//冲R角定位检测																							
	IF NOT ProductPar.iModeEN.bChamferCCDEN AND NOT ProductPar.iModeEN.bEmptyRunEN AND NOT ProductPar.iModeEN.bCcdTcpEN THEN																									
		CCD_IO.boChamferPhoto:=TRUE;																								
		fRecordMouldCCDInMainPos:=arrAxisCtrl[VirAxisNo.VirMain].Status.fActPos;																								
		fRecordMouldCCDInMainPosMod:=arrAxisCtrl[VirAxisNo.VirMain].Status.fModuloActPos;																								
		TabData[TabNo.MouldPhoto].fPhotoPosM:=fDriverDDRActPos;		
		TabData[TabNo.MouldPhoto].bCCDed_M:=TRUE;		
		TabData[TabNo.MouldPhoto].bTabOffsetNG_M:=FALSE;	
		MEMSET(ADR(CCD_COM.Chamfer),0,SIZEOF(CCD_COM.Chamfer));																		
		CCD_COM.Chamfer.iFinish:=0;																								
		iAutoAuxStep4:=10;																								
	END_IF																									
//裁切定位检测																								
	IF NOT ProductPar.iModeEN.bCuterCCDEN AND NOT ProductPar.iModeEN.bEmptyRunEN AND NOT ProductPar.iModeEN.bCcdTcpEN AND TabData[TabNo.CuterPhoto].bCCDed_M THEN																									
		CCD_IO.boCuterPhoto:=TRUE;																								
		fRecordCuterCCDInMainPos:=arrAxisCtrl[VirAxisNo.VirMain].Status.fActPos;																								
		fRecordCuterCCDInMainPosMod:=arrAxisCtrl[VirAxisNo.VirMain].Status.fModuloActPos;																								
		TabData[TabNo.CuterPhoto].fPhotoPosC:=fDriverDDRActPos;
		InteData[InteNo.Cuter-2].bIntervalFail_C:=FALSE;
		TabData[TabNo.CuterPhoto].bTabOffsetNG_C:=FALSE;	
		TabData[TabNo.CuterPhoto].bCCDed_C:=TRUE;																							
		CCD_COM.Cuter.iFinish:=0;																								
		iAutoAuxStep5:=10;																								
	END_IF																									
																				
	//************************************************************************NG踢废********************************************************************************************																									
	IF  (NOT ProductPar.iModeEN.bSizeCCDEN AND BeltData[BeltNo.NGBox1+2].fPoleNGSizeNo<>30  
		AND NOT ProductPar.iModeEN.bEmptyRunEN AND NOT ProductPar.iModeEN.bCcdTcpEN ) 		 
		OR			
	 	( BeltData[BeltNo.NGBox1+2].fPoleNGSacnNo <>30 AND NOT bFlgLineScanOver AND NOT ProductPar.iModeEN.bCcdTcpEN AND NOT ProductPar.iModeEN.bLineScanCCDEN AND NOT ProductPar.iModeEN.bEmptyRunEN)  
		OR  
		(BeltData[BeltNo.NGBox1+2].bYellowMark)  OR 
         (BeltData[BeltNo.NGBox1+2].bBlueMark)  THEN	
		NG_Sum:=NG_Sum+1;
		arrCyCtrl[EvNo.	NGPushInsideAir	].Cmd.bON:=TRUE;//踢NG料打开
		arrCyCtrl[EvNo.	NGPushInsideAir	].Cmd.bOFF:=FALSE;//踢NG料关闭		
		arrCyCtrl[EVNo.NGPushInsideVacuo].Cmd.bON:=FALSE;//踢NG料真空打开
		arrCyCtrl[EVNo.NGPushInsideVacuo].Cmd.bOFF:=TRUE;//踢NG料真空关闭																	
		BeltData[BeltNo.NGBox1+2].bHavePole:=FALSE;	
		BeltData[BeltNo.NGBox1+2].stPoleNo:='';																							
	ELSE	
		arrCyCtrl[EvNo.	NGPushInsideAir	].Cmd.bON:=FALSE;//踢NG料打开
		arrCyCtrl[EvNo.	NGPushInsideAir	].Cmd.bOFF:=TRUE;//踢NG料关闭		
		arrCyCtrl[EVNo.NGPushInsideVacuo].Cmd.bON:=TRUE;//踢NG料真空打开
		arrCyCtrl[EVNo.NGPushInsideVacuo].Cmd.bOFF:=FALSE;//踢NG料真空关闭																					
	END_IF		
												
	//iNGStep:=10;
	(*IF BeltData[BeltNo.NGBox1+2].bYellowMark THEN
		Production.NGFlag[33]:=TRUE;//感应器黄标计数;
	END_IF	*)	
																
																																																																	
(*************************************************************************裁切补偿，R角补偿计算********************************************************************************************)																									
IF NOT ProductPar.iModeEN.bEmptyRunEN AND NOT ProductPar.iModeEN.bCcdTcpEN THEN				
	(*
		//////////////////////驱动辊补偿量////////////V1////////////	
	 IF  NOT   bFlgTabPosOver THEN		
			 IF TabData[TabNo.CuterPhoto+2].bCCDed_C AND NOT TabData[TabNo.CuterPhoto+2].bTabOffsetNG_C THEN
							fDriverOffset7:=TabData[TabNo.CuterPhoto+2].fTab_OffsetC-(fDriverOffsetData[1]+fDriverOffsetData[2]);
			ELSE
						   IF ABS(fDriverOffsetData[1])<0.4 THEN
								fDriverOffset7:=fDriverOffsetData[1]*0.8;
							ELSIF ABS(fDriverOffsetData[2])<0.4 THEN
								fDriverOffset7:=fDriverOffsetData[2]*0.8;
							ELSE
								fDriverOffset7:=0;
							END_IF
			 END_IF 	
			
			IF ABS(fDriverOffset7)<10 THEN
							IF ABS(fDriverOffset7)<0.6 THEN
								Polepar.fPoleWithOffset:=LIMIT(-0.35, fDriverOffset7,0.35);
							ELSE
								Polepar.fPoleWithOffset:=fDriverOffset7;  
							END_IF
			ELSE
							IF fDriverOffset7>0 THEN
								Polepar.fPoleWithOffset:=10;
							ELSIF fDriverOffset7<0 THEN
								Polepar.fPoleWithOffset:=-10;
							END_IF	
			END_IF	

	  ELSE
					 fDriverOffset7:=fDriverOffset;
					 Polepar.fPoleWithOffset:=LIMIT(-23,fDriverOffset7,23);	
	  END_IF	
	  *)
	

	  TabData[TabNo.CuterPhoto].fTab_OffsetC;  //
	  fTab_OffsetC; //裁切下个工位反馈的极耳偏移量
		//////////////////////驱动辊补偿量////////////V1////////////			
		IF TabData[TabNo.CuterPhoto+2].bCCDed_C AND NOT TabData[TabNo.CuterPhoto+2].bTabOffsetNG_C THEN
			fDriverOffset7:=TabData[TabNo.CuterPhoto+2].fTab_OffsetC-(fDriverOffsetData[1]+fDriverOffsetData[2]);
		ELSE
			IF ABS(fDriverOffsetData[1])<0.4 THEN
				fDriverOffset7:=fDriverOffsetData[1]*0.8;
			ELSIF ABS(fDriverOffsetData[2])<0.4 THEN
				fDriverOffset7:=fDriverOffsetData[2]*0.8;
			ELSE
				fDriverOffset7:=0;
			END_IF
		END_IF 		
			
			
IF NOT 	bMA1	 THEN	
	IF  NOT   bFlgTabPosOver THEN		//计算当前片下个周期补偿量   	 
				IF ABS(fDriverOffset7)<15 THEN
								IF ABS(fDriverOffset7)<1 THEN
									//bMA1:=FALSE;
									Polepar.fPoleWithOffset:=LIMIT(-0.35, fDriverOffset7,0.35);
								ELSE
									 bMA1:=TRUE;
									 iFlgCompCount:=3;
									 iCompCount:=3;
									 arrOffset[3]:=fDriverOffset7;//+fArvDriverOffsetData ;
									 arrOffset[2]:=arrOffset[1]:=fArvDriverOffsetData;	  
									//Polepar.fPoleWithOffset:=fDriverOffset7    ;  
								END_IF		
				ELSE
								iCount20:=iCount20+1;
								 IF  ABS(fDriverOffset7)>15   AND  ABS(fDriverOffset7)<30 THEN
									  iFlgCompCount:=4;
									  iCompCount:=4;
									   bMA1:=TRUE;
									  arrOffset[4]:= SEL( fDriverOffset7>0,-15,15 )  ;
		                                                         arrOffset[3]:=SEL(fDriverOffset7>0,   fDriverOffset7+15  , fDriverOffset7-15 )  ;                         
	                                                                arrOffset[2]:=arrOffset[1]:=fArvDriverOffsetData;	  
								 ELSIF ABS(fDriverOffset7)>30   AND  ABS(fDriverOffset7)<45 THEN
									   iFlgCompCount:=5;
									   iCompCount:=5;
									    bMA1:=TRUE;
									   arrOffset[5]:=SEL( fDriverOffset7>0,-15,15 ) ;
									   arrOffset[4]:=SEL( fDriverOffset7>0,-15,15 ) ;
		                                                           arrOffset[3]:=SEL(fDriverOffset7>0,   fDriverOffset7+30  , fDriverOffset7-30 )  ;       
	                                                                    arrOffset[2]:=arrOffset[1]:=fArvDriverOffsetData;	  	
		 										 
								 ELSIF ABS(fDriverOffset7)>45   AND ABS(fDriverOffset7)<60 THEN
									   iFlgCompCount:=6;		
									    iCompCount:=6;	
									     bMA1:=TRUE;
									   arrOffset[6]:=SEL( fDriverOffset7>0,-15,15 ) ;
									   arrOffset[5]:=SEL( fDriverOffset7>0,-15,15 ) ;
									   arrOffset[4]:=SEL( fDriverOffset7>0,-15,15 ) ;									   
		                                                           arrOffset[3]:=SEL(fDriverOffset7>0,   fDriverOffset7+45  , fDriverOffset7-45 )  ;    
	                                                                  arrOffset[2]:=arrOffset[1]:=fArvDriverOffsetData;	  		 
								 ELSIF ABS(fDriverOffset7)>60   AND  ABS(fDriverOffset7)<75 THEN
									   iFlgCompCount:=7;		
									   iCompCount:=7;	
                                                                          bMA1:=TRUE;	 
									   arrOffset[7]:=SEL( fDriverOffset7>0,-15,15 ) ;
									   arrOffset[6]:=SEL( fDriverOffset7>0,-15,15 ) ;
									   arrOffset[5]:=SEL( fDriverOffset7>0,-15,15 ) ;		
									   arrOffset[4]:=SEL( fDriverOffset7>0,-15,15 ) ;						   
		                                                            arrOffset[3]:=SEL(fDriverOffset7>0,   fDriverOffset7+60  , fDriverOffset7-60 )  ;    
	                                                                   arrOffset[2]:=arrOffset[1]:=fArvDriverOffsetData;										   
								ELSIF  ABS(fDriverOffset7)>75  THEN
									   iFlgCompCount:=7;		
									   iCompCount:=7;	
                                                                           bMA1:=TRUE;	 
									   arrOffset[7]:=SEL( fDriverOffset7>0,-15,15 ) ;
									   arrOffset[6]:=SEL( fDriverOffset7>0,-15,15 ) ;
									   arrOffset[5]:=SEL( fDriverOffset7>0,-15,15 ) ;		
									   arrOffset[4]:=SEL( fDriverOffset7>0,-15,15 ) ;						   
		                                                           arrOffset[3]:=SEL(fDriverOffset7>0,   fDriverOffset7+60  , fDriverOffset7-60 )  ;    
	                                                                  arrOffset[2]:=arrOffset[1]:=fArvDriverOffsetData;		      
								 END_IF
								
				END_IF	
	ELSE	
					                       fDriverOffset7:=fDriverOffset;
								 IF  ABS(fDriverOffset7)>30   AND  ABS(fDriverOffset7)<60 THEN
									  iFlgCompCount:=4;
									  iCompCount:=4;
									   bMA1:=TRUE;
									  arrOffset[4]:= SEL( fDriverOffset7>0,-30,30 )  ;
		                                                         arrOffset[3]:=SEL(fDriverOffset7>0,   fDriverOffset7+30  , fDriverOffset7-30 )  ;                         
	                                                                arrOffset[2]:=arrOffset[1]:=fArvDriverOffsetData;	  
								 ELSIF ABS(fDriverOffset7)>60   AND  ABS(fDriverOffset7)<90 THEN
									   iFlgCompCount:=5;
									   iCompCount:=5;
									    bMA1:=TRUE;
									   arrOffset[5]:=SEL( fDriverOffset7>0,-30,30 ) ;
									   arrOffset[4]:=SEL( fDriverOffset7>0,-30,30 ) ;
		                                                           arrOffset[3]:=SEL(fDriverOffset7>0,   fDriverOffset7+60  , fDriverOffset7-60 )  ;       
	                                                                    arrOffset[2]:=arrOffset[1]:=fArvDriverOffsetData;	  	
		 										 
								 ELSIF ABS(fDriverOffset7)>90   AND ABS(fDriverOffset7)<120 THEN
									   iFlgCompCount:=6;		
									    iCompCount:=6;	
									     bMA1:=TRUE;
									   arrOffset[6]:=SEL( fDriverOffset7>0,-30,30 ) ;
									   arrOffset[5]:=SEL( fDriverOffset7>0,-30,30 ) ;
									   arrOffset[4]:=SEL( fDriverOffset7>0,-30,30 ) ;									   
		                                                           arrOffset[3]:=SEL(fDriverOffset7>0,   fDriverOffset7+90  , fDriverOffset7-90 )  ;    
	                                                                  arrOffset[2]:=arrOffset[1]:=fArvDriverOffsetData;	  		 
								 ELSIF ABS(fDriverOffset7)>120   AND  ABS(fDriverOffset7)<150 THEN
									   iFlgCompCount:=7;		
									   iCompCount:=7;	
                                                                          bMA1:=TRUE;	 
									   arrOffset[7]:=SEL( fDriverOffset7>0,-30,30 ) ;
									   arrOffset[6]:=SEL( fDriverOffset7>0,-30,30 ) ;
									   arrOffset[5]:=SEL( fDriverOffset7>0,-30,30 ) ;		
									   arrOffset[4]:=SEL( fDriverOffset7>0,-30,30 ) ;						   
		                                                            arrOffset[3]:=SEL(fDriverOffset7>0,   fDriverOffset7+120  , fDriverOffset7-120 )  ;    
	                                                                   arrOffset[2]:=arrOffset[1]:=fArvDriverOffsetData;										   
								ELSIF  ABS(fDriverOffset7)>150  THEN
						                           iFlgCompCount:=7;		
									   iCompCount:=7;	
                                                                           bMA1:=TRUE;	 
									   arrOffset[7]:=SEL( fDriverOffset7>0,-30,30 ) ;
									   arrOffset[6]:=SEL( fDriverOffset7>0,-30,30 ) ;
									   arrOffset[5]:=SEL( fDriverOffset7>0,-30,30 ) ;		
									   arrOffset[4]:=SEL( fDriverOffset7>0,-30,30 ) ;						   
		                                                            arrOffset[3]:=SEL(fDriverOffset7>0,   fDriverOffset7+120  , fDriverOffset7-120 )  ;    
	                                                                   arrOffset[2]:=arrOffset[1]:=fArvDriverOffsetData;			      
								 END_IF								 
					                //Polepar.fPoleWithOffset:=LIMIT(-23,fDriverOffset7,23);	
	 END_IF		
	 
END_IF

	(************补偿大偏移量后面的极片模糊补偿 *****************)
	IF  bMA1 THEN
		 Polepar.fPoleWithOffset:=arrOffset[iCompCount]; 
		IF 	iCompCount<=1 THEN
			bMA1:=FALSE;
			iFlgCompCount:=0;
			MEMSET(ADR(arrOffset),0,SIZEOF(arrOffset));
		END_IF
	END_IF			
		
(************计算近10次补偿有效值的平均值******************)
   K2:=0;
   fSumDriverOffsetData:=0;
	FOR i30:=1 TO 10 BY 1 DO
		IF  ABS( fDriverOffsetData[i30])  <0.3   AND  ABS( fDriverOffsetData[i30])  >0  THEN 		//
			K2:=K2+1;
		    fSumDriverOffsetData:=fSumDriverOffsetData+fDriverOffsetData[i30];
		END_IF
		
		IF  i30=10   THEN
			IF K2>=1 THEN 
			   fArvDriverOffsetData:=fSumDriverOffsetData/K2;
			ELSE
			   fArvDriverOffsetData:=0;
			END_IF
		END_IF		
	END_FOR	
	

				
(*-----------20240404
//裁切补偿计算																								
IF NOT ProductPar.iModeEN.bEmptyRunEN AND NOT ProductPar.iModeEN.bCcdTcpEN AND NOT ProductPar.iModeEN.bCuterCCDEN   THEN			
	IF   ProductPar.bCompSel OR TRUE THEN	  //极耳定位补偿方式																				
	(*	IF TabData[TabNo.CuterPhoto+2].bCCDed_C AND NOT TabData[TabNo.CuterPhoto+2].bTabOffsetNG_C THEN
			fDriverOffset7:=TabData[TabNo.CuterPhoto+2].fTab_OffsetC-(fDriverOffsetData[1]+fDriverOffsetData[2]);
		ELSE
			fDriverOffset7:=0;
		END_IF*)
		
	   
	    	 IF  NOT   bFlgTabPosOver THEN
					 
						(*IF TabData[TabNo.CuterPhoto+2].bCCDed_C AND NOT TabData[TabNo.CuterPhoto+2].bTabOffsetNG_C THEN
							fDriverOffset7:=TabData[TabNo.CuterPhoto+2].fTab_OffsetC-(fDriverOffsetData[1]+fDriverOffsetData[2]);
						ELSE
						fDriverOffset7:=0;
					  END_IF*)
			 
					 IF TabData[TabNo.CuterPhoto+2].bCCDed_C AND NOT TabData[TabNo.CuterPhoto+2].bTabOffsetNG_C THEN
							fDriverOffset7:=TabData[TabNo.CuterPhoto+2].fTab_OffsetC-(fDriverOffsetData[1]+fDriverOffsetData[2]);
					  ELSE
						   IF ABS(fDriverOffsetData[1])<0.4 THEN
								fDriverOffset7:=fDriverOffsetData[1]*0.8;
							ELSIF ABS(fDriverOffsetData[2])<0.4 THEN
								fDriverOffset7:=fDriverOffsetData[2]*0.8;
							ELSE
								fDriverOffset7:=0;
							END_IF
					  END_IF 
				  
				  
				  
                   (*   IF TabData[TabNo.CuterPhoto+2].bCCDed_C AND NOT TabData[TabNo.CuterPhoto+2].bTabOffsetNG_C THEN
							
								IF TabData[TabNo.CuterPhoto+3].bCCDed_C AND NOT TabData[TabNo.CuterPhoto+3].bTabOffsetNG_C  THEN
									fDriverOffset7:=(TabData[TabNo.CuterPhoto+2].fTab_OffsetC+TabData[TabNo.CuterPhoto+3].fTab_OffsetC)/2 - (fDriverOffsetData[1]+fDriverOffsetData[2]);
							ELSE
									fDriverOffset7:=TabData[TabNo.CuterPhoto+2].fTab_OffsetC-(fDriverOffsetData[1]+fDriverOffsetData[2]);
							END_IF
						ELSE
							IF ABS(fDriverOffsetData[1])<0.4 THEN
									fDriverOffset7:=fDriverOffsetData[1]*0.8;
								ELSIF ABS(fDriverOffsetData[2])<0.4 THEN
								fDriverOffset7:=fDriverOffsetData[2]*0.8;
							ELSE
								fDriverOffset7:=0;
								END_IF
							
						END_IF 	*)
				
					
						(*	
						IF ABS(fDriverOffset7)<10 THEN
							Polepar.fPoleWithOffset:=fDriverOffset7;
						ELSE
							IF fDriverOffset7>0 THEN
								Polepar.fPoleWithOffset:=10;
							ELSIF fDriverOffset7<0 THEN
								Polepar.fPoleWithOffset:=-10;
							END_IF	
						END_IF*)
						
								
						IF ABS(fDriverOffset7)<10 THEN
							IF ABS(fDriverOffset7)<0.6 THEN
								Polepar.fPoleWithOffset:=LIMIT(-0.35, fDriverOffset7,0.35);
							ELSE
								Polepar.fPoleWithOffset:=fDriverOffset7;  
							END_IF
						ELSE
							IF fDriverOffset7>0 THEN
								Polepar.fPoleWithOffset:=10;
							ELSIF fDriverOffset7<0 THEN
								Polepar.fPoleWithOffset:=-10;
							END_IF	
						END_IF	
				 ELSE
						  fDriverOffset7:=fDriverOffset;
						  Polepar.fPoleWithOffset:=LIMIT(-23,fDriverOffset7,23);	
				END_IF				
	ELSE//尺寸检测闭环纠偏
				 IF  NOT   bFlgTabPosOver THEN
						IF  ( BeltData[BeltNo.OverHang+1].iTabNGSizeNo=1  OR  BeltData[BeltNo.OverHang+1].iTabNGSizeNo=6 )  
							AND 0<=BeltData[BeltNo.OverHang+1].fTabSite AND BeltData[BeltNo.OverHang+1].fTabSite<90 THEN
						
							fDriverOffset7:=(PolePar.TabSitebace-BeltData[BeltNo.OverHang+1].fTabSite-fDriverOffsetData[1]-fDriverOffsetData[2]);
							
							//fDriverOffset7:=(PolePar.TabSitebace-BeltData[BeltNo.OverHang+1].fTabSite-
                                                                       //         LIMIT(-2, fDriverOffsetData[1] ,2) - LIMIT(-2, fDriverOffsetData[2] ,2)  ) ;
						ELSE
							fDriverOffset7:=0;
						END_IF		
				
						IF ABS(fDriverOffset7)<0.5 THEN
							Polepar.fPoleWithOffset:=LIMIT(-0.18,fDriverOffset7,0.18);
						ELSE
							Polepar.fPoleWithOffset:=LIMIT(-25,fDriverOffset7,25);
						END_IF
				 ELSE
						  fDriverOffset7:=fDriverOffset;
						  Polepar.fPoleWithOffset:=LIMIT(-25,fDriverOffset7,25);	
				END_IF
	END_IF
----------------20240404*)			
(*																						
	//模具前计算模具X纠偏补偿量
	IF TabData[TabNo.MouldPhoto+2].bCCDed_M AND NOT TabData[TabNo.MouldPhoto+2].bTabOffsetNG_M AND NOT ProductPar.iModeEN.bMouldXOffsetEN THEN
		fMouldXOffset7:=TabData[TabNo.MouldPhoto+2].fTab_OffsetM-(fDriverOffsetData[1]+fDriverOffsetData[2]+fDriverOffsetData[3]);
	ELSE
		fMouldXOffset7:=0;
	END_IF
*)	
	//模具前计算模具X纠偏补偿量	
	
	(*
	IF TabData[TabNo.MouldPhoto+2].bCCDed_M AND NOT TabData[TabNo.MouldPhoto+2].bTabOffsetNG_M AND NOT ProductPar.iModeEN.bMouldXOffsetEN THEN
		fMouldXOffset7:=TabData[TabNo.MouldPhoto+2].fTab_OffsetM-(fDriverOffsetData[1]+fDriverOffsetData[2]+fDriverOffsetData[3]);
	ELSE
		fMouldXOffset7:=0;
	END_IF	*)
										(*****************************R角补偿****************************************)	
     IF TabData[TabNo.MouldPhoto+2].bCCDed_M AND NOT TabData[TabNo.MouldPhoto+2].bTabOffsetNG_M AND NOT ProductPar.iModeEN.bMouldXOffsetEN THEN
		fMouldXOffset7:=TabData[TabNo.MouldPhoto+2].fTab_OffsetM-
                                             ( LIMIT( -1,  fDriverOffsetData[1] ,1 ) + LIMIT( -1,  fDriverOffsetData[2] ,1)+ LIMIT( -1,  fDriverOffsetData[3] ,1)  );
	ELSE
		fMouldXOffset7:=0;
	END_IF	
	
    IF TabData[TabNo.MouldPhoto+2].bCCDed_M AND NOT TabData[TabNo.MouldPhoto+2].bTabOffsetNG_M AND NOT ProductPar.iModeEN.bMouldXOffsetEN THEN
		fMouldXOffset8:= TabData[TabNo.MouldPhoto+2].fTab_OffsetY ;
                                         
	ELSE
		
		IF  NOT TabData[TabNo.MouldPhoto+3].bTabOffsetNG_M THEN
		    fMouldXOffset8:= TabData[TabNo.MouldPhoto+3].fTab_OffsetY ;
		ELSIF NOT TabData[TabNo.MouldPhoto+4].bTabOffsetNG_M THEN
			fMouldXOffset8:= TabData[TabNo.MouldPhoto+4].fTab_OffsetY ;
		ELSE
			fMouldXOffset8:=0;
		END_IF
			
	END_IF	 
	
	
	
	
	
	IF NOT ProductPar.iModeEN.bMouldXclosureEN AND NOT bCyDDRMark THEN
		IF iRTransCompCount=1  THEN
			iRTransCompCount:=28;
			(************计算近10次R角横深有效值的平均值******************)
		   K4:=0;
		   fSumTransverData:=0;
			FOR i30:=3 TO 22 BY 1 DO
				IF iPartSelect=1 THEN//正极      2---4
					IF BeltData[i30].fPoleNGSizeNo=30 THEN
						K4:=K4+1;
						(*正极RoundedSize7为叠片侧、RoundedSize8为切刀侧，故RoundedSize7-RoundedSize8*)	
						fSumTransverData:=fSumTransverData+(BeltData[i30].RoundedSize7-BeltData[i30].RoundedSize8)/2;			
					END_IF
				ELSE//负极     1.8----3.8
					IF BeltData[i30].fPoleNGSizeNo=30 THEN
						K4:=K4+1;
						(*负极RoundedSize8为叠片侧、RoundedSize7为切刀侧，故RoundedSize8-RoundedSize7*)	
						fSumTransverData:=fSumTransverData+(BeltData[i30].RoundedSize8-BeltData[i30].RoundedSize7)/2;				
					END_IF			
				END_IF		
		
				IF  i30=22   THEN
					IF K4>=15 THEN 
					  // fArvTransverData:=fArvTransverData+LIMIT(-0.1,fSumTransverData/K4*0.3,0.1);  //(-0.25,fSumTransverData/K4*0.3,0.25)
					   fArvTransverData:=fArvTransverData+SEL( ABS(fSumTransverData/K4)>=0.1,0,LIMIT(-0.25,fSumTransverData/K4*0.3,0.25));
					ELSE
					   fArvTransverData:=0;//???
					END_IF
				END_IF		
			END_FOR		
		END_IF
		IF iRTransCompCount>=1 THEN	
			iRTransCompCount:=iRTransCompCount-1;
		END_IF
	ELSE
		iRTransCompCount:=28;
		fArvTransverData:=0;	
	END_IF

	
	
	(***************************R角纵深闭环**********************************)
	bComMode:=TRUE;
IF NOT ProductPar.iModeEN.bMouldYclosureEN AND NOT bCyDDRMark THEN
	
 IF iRTransCompCount2=1  THEN
			iRTransCompCount2:=28;
			
			(************计算近10次R角纵深有效值的平均中值******************)
		   K3:=0;
		   fSumTransverData2:=0;
	FOR i30:=3 TO 22 BY 1 DO
									
			IF NOT bComMode THEN  //纵深
				(*
				IF iPartSelect=1 THEN//正极             4.7----6.3  
					(*   V1 角纵深       正极RoundedSize3为叠片侧R角纵深    、RoundedSize4为切刀侧R角纵深 ，RoundedSize3+RoundedSize4    *)
	                 IF 4.7<=BeltData[i30].RoundedSize3   AND  BeltData[i30].RoundedSize4<=6.3 THEN 
				         fSumTransverData:=fSumTransverData+(BeltData[i30].RoundedSize3+BeltData[i30].RoundedSize4)/2;		
						 K3:=K3+1;
					END_IF				
				ELSIF  iPartSelect=2 THEN//负极        1.8----3.4
					(*   V1 角纵深       正极RoundedSize3为叠片侧R角纵深    、RoundedSize4为切刀侧R角纵深 ，RoundedSize3+RoundedSize4    *)
	                 IF 1.8<=BeltData[i30].RoundedSize3   AND  BeltData[i30].RoundedSize4<=3.4 THEN 
				         fSumTransverData:=fSumTransverData+(BeltData[i30].RoundedSize3+BeltData[i30].RoundedSize4)/2;		
						 K3:=K3+1;
					END_IF			
			   END_IF
				*)
               ;	
		   ELSE//面积
				IF iPartSelect=1 THEN//正极             C+D=32.972   
				   (*   V2角面积     正极RoundedSize1为叠片侧R角面积  、RoundedSize2为切刀侧R角面积 ，RoundedSize3+RoundedSize4    *)	
				   (* IF BeltData[i30].fPoleNGSizeNo=30   THEN 	
					    fSumTransverData2:=fSumTransverData2+( (BeltData[i30].RoundedSize1+BeltData[i30].RoundedSize2)-32.972 );	
					    K3:=K3+1;
					END_IF*)	
				    IF BeltData[i30].fPoleNGSizeNo=30   THEN 	
					    fSumTransverData2:=fSumTransverData2+(BeltData[i30].RoundedSize1+BeltData[i30].RoundedSize2);	
					    K3:=K3+1;
					END_IF					
					
				ELSIF  iPartSelect=2 THEN//负极     //C+D=11.608   //C+D=11.877
				   (*   V2角面积     正极RoundedSize1为叠片侧R角面积  、RoundedSize2为切刀侧R角面积 ，RoundedSize3+RoundedSize4    *)	
				   (* IF BeltData[i30].fPoleNGSizeNo=30THEN 	
					    fSumTransverData2:=fSumTransverData2+( (BeltData[i30].RoundedSize1+BeltData[i30].RoundedSize2)-11.877 );	
					    K3:=K3+1;
					END_IF*)		
				    IF BeltData[i30].fPoleNGSizeNo=30THEN 	
					    fSumTransverData2:=fSumTransverData2+(BeltData[i30].RoundedSize1+BeltData[i30].RoundedSize2);	
					    K3:=K3+1;
					END_IF						
				END_IF	
			END_IF
							
				IF  i30=22  THEN
					IF  iPartSelect=1 THEN//正极  
							IF K3>=15 THEN 
								IF NOT bComMode THEN  //V1 角纵深    补偿方式
									(*fArvTransverData2:=fArvTransverData2+LIMIT( -0.1,   fSumTransverData2/K3-fRSizeBase   , 0.1 )  ;*)
									;
								ELSE    //V2 角面积  补偿方式
									//fArvTransverData2:=fSumTransverData2/K3;
									//   fArvTransverData2:=fArvTransverData2+LIMIT(-0.25,fSumTransverData2/K3*0.3,0.25);
								    //fArvTransverData2:=SEL( ABS(fSumTransverData2/K3-32.972)>=1.2 ,0 ,fArvTransverData2+LIMIT(-0.1,(fSumTransverData2/K3-32.972)*0.3,0.1));
									 IF ABS(fSumTransverData2/K3-32.972)>=1.2 THEN
										fArvTransverData2:=fArvTransverData2+LIMIT(-0.1,(fSumTransverData2/K3-32.972)*0.3,0.1); 
									 END_IF
									
									
								END_IF		   
							ELSE
							   fArvTransverData2:=0;
							END_IF
					ELSIF  iPartSelect=2 THEN//负极  
								IF K3>=15 THEN 
									IF NOT bComMode THEN  //V1 角纵深    补偿方式
										(*fArvTransverData2:=fArvTransverData2+LIMIT( -0.1,   fSumTransverData2/K3-fRSizeBase   , 0.1 )  ;*)
										;
									ELSE    //V2 角面积  补偿方式
										//fArvTransverData2:=fSumTransverData2/K3;
										//   fArvTransverData2:=fArvTransverData2+LIMIT(-0.25,fSumTransverData2/K3*0.3,0.25);
										//fArvTransverData2:=SEL( ABS(fSumTransverData2/K3-11.877)>=0.55 ,0 ,fArvTransverData2+LIMIT(-0.1,(fSumTransverData2/K3-11.877)*0.3,0.1));
										IF ABS(fSumTransverData2/K3-11.877)>=0.55 THEN
											fArvTransverData2:=fArvTransverData2+LIMIT(-0.1,(fSumTransverData2/K3-11.877)*0.3,0.1);
										END_IF
									END_IF		   
							ELSE
							   fArvTransverData2:=0;
							END_IF						
					END_IF		
				END_IF	
				
		END_FOR		
			
	END_IF	
		
		IF iRTransCompCount2>=1 THEN	
			iRTransCompCount2:=iRTransCompCount2-1;
		END_IF
		
ELSE
		iRTransCompCount2:=28;
		fArvTransverData2:=0;	
END_IF
	
	
	
	
	
	
	
	IF arrAxisPar[AxisNo.MouldRectify_X].arrTargetPoint[1]-fMouldXOffset7>arrAxisPar[AxisNo.MouldRectify_X].arrTargetPoint[3] OR
		arrAxisPar[AxisNo.MouldRectify_X].arrTargetPoint[1]-fMouldXOffset7<arrAxisPar[AxisNo.MouldRectify_X].arrTargetPoint[4] AND NOT ProductPar.iModeEN.bMouldXOffsetEN 
	THEN
		Polepar.fMouldX_Offset:=arrAxisPar[AxisNo.MouldRectify_X].arrTargetPoint[1]-arrAxisCtrl[AxisNo.MouldRectify_X].Status.fSetPos;
		stAlarm.arrLightWarn[8]:=TRUE;//模具X补偿量超过纠偏电机行程
	ELSE
		Polepar.fMouldX_Offset:=fMouldXOffset7;
	END_IF
	
	//arrAxisPar[AxisNo.MouldRectify_X].arrTargetPoint[2]:=arrAxisPar[AxisNo.MouldRectify_X].arrTargetPoint[1]+fArvTransverData-Polepar.fMouldX_Offset;   //V1
	
	                            //TabData[TabNo.MouldPhoto+2].fTab_OffsetM
	//arrAxisPar[AxisNo.MouldRectify_Y].arrTargetPoint[2]:=arrAxisPar[AxisNo.MouldRectify_Y].arrTargetPoint[1]-  (TabData[TabNo.MouldPhoto+2].fTab_OffsetM + TabData[TabNo.MouldPhoto+2].fTab_OffsetM )/2     ;   //V1
								
	
(*	
  IF   NOT CutMark_R[0] THEN
	arrAxisPar[AxisNo.MouldRectify_X].arrTargetPoint[2]:=arrAxisPar[AxisNo.MouldRectify_X].arrTargetPoint[1]-Polepar.fMouldX_Offset;
  ELSE
      arrAxisPar[AxisNo.MouldRectify_X].arrTargetPoint[2]:=arrAxisPar[AxisNo.MouldRectify_X].arrTargetPoint[1];
 END_IF		
*)   //V2		


(*
  IF  ABS(   PolePar.TabSitebace-BeltData[BeltNo.OverHang+1].fTabSite )<=4    AND     BeltData[BeltNo.OverHang+1].iTabNGSizeNo=1    THEN
	arrAxisPar[AxisNo.MouldRectify_X].arrTargetPoint[2]:=arrAxisPar[AxisNo.MouldRectify_X].arrTargetPoint[1]-Polepar.fMouldX_Offset;
  ELSE
      arrAxisPar[AxisNo.MouldRectify_X].arrTargetPoint[2]:=arrAxisPar[AxisNo.MouldRectify_X].arrTargetPoint[1];
 END_IF	
*)//V3



	
ELSE
	Polepar.fPoleWithOffset:=0;
	Polepar.fMouldX_Offset:=0;
END_IF	
																						
//记录模具，切刀当前的凸轮																								
	iMouldRunTableSel:=fbMouldCam.iTableSel;																									
	iCuterRunTableSel:=fbCuterCam.iTableSel;																									
	iAutoRunStep:=4015;		

	(*************************************************************************黄标位置判断*******************************************************************************************)	
4015: 
	//	PolePar.YellScope;//黄标检测有效范围,,mm	------R角
	FOR i8:=20 TO 1 BY -1 DO	
		IF ( PolePar.fPoleWidth-PolePar.fYellowBreadth<=(aYellowPos[i8]+PolePar.fBlue_Mould-fDriverDDRActPos)  )    AND
		    (  ( aYellowPos[i8]+PolePar.fBlue_Mould-fDriverDDRActPos)<=PolePar.fPoleWidth+PolePar.fYellowBreadth  )  AND  
			aYellowPos[i8]>0 THEN
			aYellowJump_R[1]:=TRUE;//极片黄标R角跳切标志
			aYellowMark[1]:=TRUE;//第1片黄标
			aYellowPos_R[1]:=aYellowPos[i8]+PolePar.fBlue_Mould-fDriverDDRActPos;
			Production.NGFlag[44]:=TRUE;//黄黄标跳切计数
			//Production.NGFlag[45]:=TRUE;//黄黄标计数
			EXIT;		
		END_IF			
	END_FOR
	
	FOR i21:=20 TO 1 BY -1 DO	
		IF aYellowPos[i21]+PolePar.fBlue_Mould-fDriverDDRActPos < PolePar.fPoleWidth  AND  aYellowPos[i21]+PolePar.fBlue_Mould-fDriverDDRActPos>0  THEN
			aYellowMark[1]:=TRUE;//第1片黄标
			EXIT;		
		END_IF
	END_FOR
		
	//	PolePar.YellScope;//黄标检测有效范围,,mm	------裁切
	FOR i9:=20 TO 1 BY -1 DO	
		IF (PolePar.fPoleWidth-PolePar.fYellowBreadth<=(aYellowPos[i9]+PolePar.fBlue_Mould+5*PolePar.fPoleWidth-fDriverDDRActPos ))
			AND ( (aYellowPos[i9]+PolePar.fBlue_Mould+5*PolePar.fPoleWidth-fDriverDDRActPos)<=PolePar.fPoleWidth+PolePar.fYellowBreadth )
			AND aYellowPos[i9]>0 THEN						
			aYellowJump_C[1]:=TRUE;//极片黄标R角跳切标志
			aYellowPos_C[1]:=aYellowPos[i9]+PolePar.fBlue_Mould+5*PolePar.fPoleWidth-fDriverDDRActPos;
			//aYellowPos[i9]:=0;
			EXIT;
		END_IF
	END_FOR	
	
	FOR i9:=20 TO 1 BY -1 DO	//清除超范围黄标位置
		IF  ( ((aYellowPos[i9]+PolePar.fBlue_Mould+5*PolePar.fPoleWidth-fDriverDDRActPos ) <= -(PolePar.fPoleWidth+100)     )  OR 
			(ABS(aYellowPos[i9]-fDriverDDRActPos)>=PolePar.fBlue_Mould+5*PolePar.fPoleWidth+200)  )
			AND aYellowPos[i9]>0 THEN						
			aYellowPos[i9]:=0;
		END_IF
	END_FOR		
	
    FOR i9:=20 TO 2 BY -1 DO	//清除超范围置差很小的值
		IF ABS (aYellowPos[i9]- aYellowPos[i9-1] )<=6 
		   AND aYellowPos[i9]>0 AND aYellowPos[i9-1]>0   THEN						
			aYellowPos[i9]:=(aYellowPos[i9]+ aYellowPos[i9-1])/2 ;
			aYellowPos[i9-1]:= 0  ;
		END_IF
	END_FOR		
	
	
	FOR i9:=20 TO 1 BY -1 DO	 //输出黄标到裁切的距离    同时输出皮带上黄标MACK标志
		IF   aYellowPos[i9]>0 THEN						
			  aYellowPos_R2[i9]:=aYellowPos[i9]+PolePar.fBlue_Mould+5*PolePar.fPoleWidth-fDriverDDRActPos;
		ELSE
	        aYellowPos_R2[i9]:=0;
		END_IF
	END_FOR		
	
	(*********************************************接带处理****************************************************)
	FOR i8:=20 TO 1 BY -1 DO	 //-----R角
		IF ( PolePar.fPoleWidth-160<=(aTapePos[i8]+PolePar.fTape_Mould-fDriverDDRActPos)  )    AND
		    (  ( aTapePos[i8]+PolePar.fTape_Mould-fDriverDDRActPos)<=PolePar.fPoleWidth+160  )  AND  
			aTapePos[i8]>0 THEN
			aTapeJump_R[1]:=TRUE;//极片接带R角跳切标志
			aTapeMark[1]:=TRUE;//第1片黄标
			EXIT;		
		END_IF			
	END_FOR
	
	FOR i9:=20 TO 1 BY -1 DO	 	//		------裁切
		IF (PolePar.fPoleWidth-160<=(aTapePos[i9]+PolePar.fTape_Mould+5*PolePar.fPoleWidth-fDriverDDRActPos ))
			AND ( (aTapePos[i9]+PolePar.fTape_Mould+5*PolePar.fPoleWidth-fDriverDDRActPos)<=PolePar.fPoleWidth+160 )
			AND aTapePos[i9]>0 THEN						
			aTapeJump_C[1]:=TRUE;//极片接带跳切标志
			EXIT;
		END_IF
	END_FOR	
	
	FOR i9:=20 TO 1 BY -1 DO	//清除超范围黄标位置
		IF  ( ((aTapePos[i9]+PolePar.fTape_Mould+5*PolePar.fPoleWidth-fDriverDDRActPos ) <= -(PolePar.fPoleWidth+100)     )  OR 
			(ABS(aTapePos[i9]-fDriverDDRActPos)>=PolePar.fTape_Mould+5*PolePar.fPoleWidth+200)  )
			AND aTapePos[i9]>0 THEN						
			aTapePos[i9]:=0;
		END_IF
	END_FOR		
	
    FOR i9:=20 TO 2 BY -1 DO	//清除超范围置差很小的值
		IF ABS (aTapePos[i9]- aTapePos[i9-1] )<=8 
		   AND aTapePos[i9]>0 AND aTapePos[i9-1]>0   THEN						
			aTapePos[i9]:=(aTapePos[i9]+ aTapePos[i9-1])/2 ;
			aTapePos[i9-1]:=0  ;
		END_IF
	END_FOR	
	
	FOR i9:=20 TO 1 BY -1 DO	 //输出黄标到裁切的距离    同时输出皮带上黄标MACK标志
		IF   aTapePos[i9]>0 THEN						
			  aTapePos_R2[i9]:=aTapePos[i9]+PolePar.fTape_Mould+5*PolePar.fPoleWidth-fDriverDDRActPos;
	    ELSE
			  aTapePos_R2[i9]:=0;
		END_IF
	END_FOR	

	iAutoRunStep:=4020;		
		
(*************************************************************************裁切角度补偿计算*******************************************************************************************)																
4020://																	
////////////////////裁切前计算裁切角度纠偏量//////////////////////////正极:CCD发正值，意指角度纠偏往逆时针转	,而电机JOG+为顺时针，故初始位置减纠偏量   
                                                                       //            	负极:CCD发正值，意指角度纠偏往顺时针转,而电机JOG+为逆时针，故初始位置减纠偏量																									
	IF NOT ProductPar.iModeEN.bEmptyRunEN AND NOT ProductPar.iModeEN.bDegreeRecEN THEN																	
		fDegreeRec1:=FC_Variance(fOffsetDeg);						//方差只能体现偏移大小。																		
	ELSE																									
		fDegreeRec1:=0;																								
	END_IF																									
	IF fDegreeRec1>=0.005 AND NOT ProductPar.iModeEN.bEmptyRunEN THEN   //方差大于0.05  相当于偏差值-平均值达到了0.1°																									
		fDegreeRec2:=(fOffsetDeg[1]+fOffsetDeg[2]+fOffsetDeg[3]+fOffsetDeg[4]+fOffsetDeg[5]+fOffsetDeg[6]+fOffsetDeg[7]+fOffsetDeg[8])/8;
	ELSE
		fDegreeRec2:=Polepar.fDegreeRectify;//	方差小于门槛值，取上次的纠偏量																						
	END_IF			
																						
	IF NOT ProductPar.iModeEN.bEmptyRunEN AND NOT ProductPar.iModeEN.bDegreeRecEN  AND FALSE     THEN	
		IF arrAxisPar[AxisNo.CuterDegRectify].arrTargetPoint[1]-fDegreeRec2> arrAxisPar[AxisNo.CuterDegRectify].arrTargetPoint[3] OR 
			arrAxisPar[AxisNo.CuterDegRectify].arrTargetPoint[1]-fDegreeRec2< arrAxisPar[AxisNo.CuterDegRectify].arrTargetPoint[4] THEN	
																							
			  Polepar.fDegreeRectify:=arrAxisPar[AxisNo.CuterDegRectify].arrTargetPoint[1]-arrAxisCtrl[AxisNo.CuterDegRectify].Status.fSetPos;
			  stAlarm.arrLightWarn[9]:=TRUE;//裁切角度纠偏量超过纠偏电机行程																										
		ELSE
			Polepar.fDegreeRectify:=fDegreeRec2;	
			MEMSET(ADR(fOffsetDeg),0,SIZEOF(fOffsetDeg));
		END_IF	
		arrAxisPar[AxisNo.CuterDegRectify].arrTargetPoint[2]:=arrAxisPar[AxisNo.CuterDegRectify].arrTargetPoint[1]-Polepar.fDegreeRectify;																																											
	ELSE																									
		arrAxisPar[AxisNo.CuterDegRectify].arrTargetPoint[2]:=arrAxisPar[AxisNo.CuterDegRectify].arrTargetPoint[1];																								
	END_IF		

(*************************************************************************凸轮切换*******************************************************************************************)
//模具凸轮判断			
	IF ((*InteData[InteNo.Mould-1].bBlueNG OR*)  aYellowJump_R[1]   OR   aTapeJump_R[1]  OR bCyDDRMark  )         THEN		// AND NOT ProductPar.iModeEN.bEmptyRunEN     CutMark_R[2]  OR
		iCount10:=	iCount10+1;		   																		
		IF iMouldRunTableSel=1 THEN																								
			fbMouldCam.iTableSel:=2;																							
		ELSE																					
			fbMouldCam.iTableSel:=3; 																							
		END_IF;//模具凸轮切换为stop																								
	ELSE																									
		fbMouldCam.iTableSel:=1; //模具凸轮切换为正常																								
	END_IF		
																				
//裁切凸轮判断	
	IF (InteData[InteNo.Cuter-1].bLineScanNG AND NOT ProductPar.iModeEN.bLineScanCCDEN) OR aYellowJump_C[1]  OR   aTapeJump_C[1]        THEN		 //(*InteData[InteNo.Cuter-1].bBlueNG AND NOT ProductPar.iModeEN.bFlgBlueEN) OR *)																							
		IF iCuterRunTableSel=1 THEN																								
			fbCuterCam.iTableSel:=2;																							
		ELSE																								
			fbCuterCam.iTableSel:=3; 																							
		END_IF;//裁切凸轮切换为stop																								
	ELSE																									
			fbCuterCam.iTableSel:=1;//裁切凸轮切换为正常																								
	END_IF
																
(*************************************************************************补偿值更新*****************************************************************************************)		
	IF   ProductPar.bCompSel THEN		
		IF NOT ProductPar.iModeEN.bEmptyRunEN AND NOT ProductPar.iModeEN.bCcdTcpEN AND NOT ProductPar.iModeEN.bCuterOffsetEN THEN																									
			fbDriverCam.fCompensation:=Polepar.fPoleWithOffset;////修改关键点																								
		ELSE																									
			fbDriverCam.fCompensation:=0;//不修改关键点																								
		END_IF																									
																												
		IF NOT ProductPar.iModeEN.bEmptyRunEN AND NOT ProductPar.iModeEN.bCcdTcpEN AND NOT ProductPar.iModeEN.bCuterOffsetEN THEN																									
			fPoleBufferCompensation:=Polepar.fPoleWithOffset;																								
			fbUwindTen.fCompensation:=SEL(fbCuterCam.iTableSel=1,fDriverOffsetData[1],Polepar.fPoleWithOffset);																											
			fbAuxDriverTen.fCompensation:=Polepar.fPoleWithOffset;																								
		ELSE																									
			fPoleBufferCompensation:=0;																								
			fbUwindTen.fCompensation:=0;																						
			fbAuxDriverTen.fCompensation:=0;																								
		END_IF		
	ELSE
		  IF  NOT   bFlgTabPosOver THEN
					IF NOT ProductPar.iModeEN.bEmptyRunEN AND NOT ProductPar.iModeEN.bCcdTcpEN AND NOT ProductPar.iModeEN.bCuterOffsetEN  THEN	//AND fbCuterCam.iTableSel=1		
						//fbDriverCam.fCompensation:=SEL(fbCuterCam.iTableSel=1 ,fDriverOffsetData[1],Polepar.fPoleWithOffset);	////修改关键点																												
						fbDriverCam.fCompensation:=SEL(fbCuterCam.iTableSel=1 AND PolePar.TabSitebace<>BeltData[BeltNo.OverHang+1].fTabSite ,SEL(ABS(fDriverOffsetData[1])<0.18,0,fDriverOffsetData[1]),Polepar.fPoleWithOffset);	////修改关键点																										
					ELSE
						fbDriverCam.fCompensation:=0;//不修改关键点																								
					END_IF																															
				//////////////////////极片缓存凸轮缩放,放卷张力&辅驱张力缩放///////////////////////																										
					IF NOT ProductPar.iModeEN.bEmptyRunEN AND NOT ProductPar.iModeEN.bCcdTcpEN AND NOT ProductPar.iModeEN.bCuterOffsetEN  THEN		//AND fbCuterCam.iTableSel=1																							
						fPoleBufferCompensation:=SEL(fbCuterCam.iTableSel=1 AND PolePar.TabSitebace<>BeltData[BeltNo.OverHang+1].fTabSite ,SEL(ABS(fDriverOffsetData[1])<0.18,0,fDriverOffsetData[1]),Polepar.fPoleWithOffset);																							
						fbUwindTen.fCompensation:=SEL(fbCuterCam.iTableSel=1 AND PolePar.TabSitebace<>BeltData[BeltNo.OverHang+1].fTabSite ,SEL(ABS(fDriverOffsetData[1])<0.18,0,fDriverOffsetData[1]),Polepar.fPoleWithOffset);																						
						fbAuxDriverTen.fCompensation:=SEL(fbCuterCam.iTableSel=1 AND PolePar.TabSitebace<>BeltData[BeltNo.OverHang+1].fTabSite ,SEL(ABS(fDriverOffsetData[1])<0.18,0,fDriverOffsetData[1]),Polepar.fPoleWithOffset);																						
					ELSE																									
						fPoleBufferCompensation:=0;																								
						fbUwindTen.fCompensation:=0;																								
						fbAuxDriverTen.fCompensation:=0;																								
					END_IF	
		 ELSE
			IF NOT ProductPar.iModeEN.bEmptyRunEN AND NOT ProductPar.iModeEN.bCcdTcpEN AND NOT ProductPar.iModeEN.bCuterOffsetEN THEN																									
					fPoleBufferCompensation:=Polepar.fPoleWithOffset;																								
					fbUwindTen.fCompensation:=Polepar.fPoleWithOffset;																											
					fbAuxDriverTen.fCompensation:=Polepar.fPoleWithOffset;			
			   fbDriverCam.fCompensation:=Polepar.fPoleWithOffset;////修改关键点																								
				ELSE																									
					fPoleBufferCompensation:=0;																								
					fbUwindTen.fCompensation:=0;																						
					fbAuxDriverTen.fCompensation:=0;				
					  fbDriverCam.fCompensation:=0;////修改关键点																			
			END_IF	
		
		END_IF		
	END_IF
	

	//////////////////////模具前CCD检测计算极耳间距////////////////////////																								
			IF TabData[TabNo.MouldPhoto+1].bCCDed_M AND TabData[TabNo.MouldPhoto+2].bCCDed_M AND NOT TabData[TabNo.MouldPhoto+1].bTabOffsetNG_M AND NOT TabData[TabNo.MouldPhoto+2].bTabOffsetNG_M THEN																									
				fTabInteM_1:=PolePar.fPoleWidth+fDriverOffsetData[2]+(TabData[TabNo.MouldPhoto+1].fTab_OffsetM-TabData[TabNo.MouldPhoto+2].fTab_OffsetM);																								
			ELSE																									
				fTabInteM_1:=PolePar.fPoleWidth;																								
			END_IF																																																		
			InteData[InteNo.Mould-1].fTabIntervalM:=fTabInteM_1;																								
		
			IF TabData[TabNo.MouldPhoto+1].fPhotoPosM>TabData[TabNo.MouldPhoto+2].fPhotoPosM AND TabData[TabNo.MouldPhoto+1].bCCDed_M AND TabData[TabNo.MouldPhoto+2].bCCDed_M AND NOT TabData[TabNo.MouldPhoto+1].bTabOffsetNG_M AND NOT TabData[TabNo.MouldPhoto+2].bTabOffsetNG_M THEN																									
				fTabInteM_2:=TabData[TabNo.MouldPhoto+1].fPhotoPosM-TabData[TabNo.MouldPhoto+2].fPhotoPosM+(TabData[TabNo.MouldPhoto+2].fTab_OffsetM-TabData[TabNo.MouldPhoto+1].fTab_OffsetM);																								
			ELSE																									
				fTabInteM_2:=PolePar.fPoleWidth;																								
			END_IF																																																																						
		//////////////////////模具前极耳间距内前后肩宽状况判断////////////////////////	
			IF NOT ProductPar.iModeEN.bMouldXOffsetEN THEN																										
				IF ABS(InteData[InteNo.Mould-1].fTabIntervalM-PolePar.fPoleWidth)<=0.5 THEN//片宽偏差小于等于0.5																									
					InteData[InteNo.Mould-1].bTabInteFr_M:=FALSE;																								
					InteData[InteNo.Mould-1].bTabInteBe_M:=FALSE;																								
				ELSE																									
					IF NOT InteData[InteNo.Mould].bTabInteBe_M THEN																								
						InteData[InteNo.Mould-1].bTabInteFr_M:=FALSE;																							
						InteData[InteNo.Mould-1].bTabInteBe_M:=TRUE;																							
					ELSE																								
						InteData[InteNo.Mould-1].bTabInteFr_M:=TRUE;																							
						InteData[InteNo.Mould-1].bTabInteBe_M:=FALSE;																							
					END_IF																								
				END_IF		
			END_IF																							
		
			FOR i1:=1 TO 50 BY 1 DO 																									
					IF i1<50 THEN 																							
						 fM_TabInterData[51-i1]:=fM_TabInterData[50-i1];																																											
					ELSE																							
						fM_TabInterData[1]:=fTabInteM_1;																																											
					END_IF; 																							
			END_FOR; 
	FOR i1:=1 TO 50 BY 1 DO //主驱补偿值记录																									
		IF i1<50 THEN 																							
		   	fDriverOffsetData[51-i1]:=fDriverOffsetData[50-i1];																																											
		ELSIF   ProductPar.bCompSel THEN																						
			fDriverOffsetData[1]:=Polepar.fPoleWithOffset;	//裁切定位补偿
		ELSE
			fDriverOffsetData[1]:=fPoleBufferCompensation;//尺寸检测闭环补偿																																										
		END_IF; 																							
	END_FOR; 	
	 IF     iCompCount>=1 THEN	
            iCompCount:=iCompCount-1;
     END_IF																																																													
	iAutoRunStep:=4050;		


4050:	
(*
	IF stAlarm.arrFlowAlarm[35] OR stAlarm.arrFlowAlarm[37] OR stAlarm.arrFlowAlarm[38] THEN
		iAutoRunStep:=500;
		;
	ELSIF arrAxisCtrl[VirAxisNo.VirMain].Status.fModuloActPos>=310 THEN																	
		iAutoRunStep:=350;	
	END_IF	
	
*)

	IF arrAxisCtrl[VirAxisNo.VirMain].Status.fModuloActPos>=300 THEN																	
		iAutoRunStep:=4060;	
	END_IF		
	
	Production.OutFlag1:=FALSE;//产能计数
	Production.OutFlag2:=FALSE;//产能计数
	FOR i:=1 TO 50 DO//NG类型标志位复位
		Production.NGFlag[i]:=FALSE;
	END_FOR		

4060:
 IF ProductPar.iLineScanSel THEN
    IF  bFlgLineScanOver  THEN  //通讯线扫超240周期给结果      数据移位需要单独处理
		
			  //上线扫结果判断	
				FOR i1:=1 TO 20 BY 1 DO 																									
					IF i1<20 THEN 																							
						 XianSaong_Up[20-i1]:=XianSaong_Up[19-i1];																						
					ELSE																				
						XianSaong_Up[0]:=CCD_COM.Scan.iResult_UP;																											
					END_IF; 																							
				 END_FOR; 
		
			//下线扫结果判断	
				FOR i1:=1 TO 20 BY 1 DO 																									
					IF i1<20 THEN 																							
						 XianSaong_Down[20-i1]:=XianSaong_Down[19-i1];																						
					ELSE																						
						XianSaong_Down[0]:= CCD_COM.Scan.iResult_Down;																									
					END_IF; 																							
				 END_FOR;
				 
				
          	     IF XianSaong_Down[0]=30 AND XianSaong_Up[1]=30 THEN//---------------------------------线扫OK结果由8改为30，，，CCD需要同步更改
					    BeltData[BeltNo.NGBox1+2].fPoleNGSacnNo:=30; //线扫NG类型
			    ELSE
					//剔废前一工位汇总结果，5号位置，，，，，剔废工位为6
						IF XianSaong_Down[0]<>30 AND XianSaong_Up[1]=30 THEN
							BeltData[BeltNo.NGBox1+2].fPoleNGSacnNo:=XianSaong_Down[0];
						END_IF
		
						IF XianSaong_Down[0]=30 AND XianSaong_Up[1]<>30 THEN
							BeltData[BeltNo.NGBox1+2].fPoleNGSacnNo:=XianSaong_Up[1];
						END_IF
		
						IF XianSaong_Down[0]<>30 AND XianSaong_Up[1]<>30 THEN
							BeltData[BeltNo.NGBox1+2].fPoleNGSacnNo:=XianSaong_Up[1];
						END_IF				
		        END_IF	
			
			IF CCD_COM.Scan.iResult_UP=33 AND NOT ProductPar.iModeEN.bCcdTcpEN AND NOT ProductPar.iModeEN.bLineScanCCDEN THEN
				fDA1:=        arrAxisCtrl[VirAxisNo.VirMain].Status.fModuloActPos;
				stAlarm.arrFlowAlarm[25]:=TRUE;//上线扫超时报警
			END_IF	
			IF CCD_COM.Scan.iResult_Down=33 AND NOT ProductPar.iModeEN.bCcdTcpEN AND NOT ProductPar.iModeEN.bLineScanCCDEN THEN
				fDA2:=        arrAxisCtrl[VirAxisNo.VirMain].Status.fModuloActPos;
				stAlarm.arrFlowAlarm[27]:=TRUE;//下线扫超时报警
			END_IF	
	(*
			IF  CCD_COM.Scan.iResult_UP<>33 AND CCD_COM.Scan.iResult_Down<>33 THEN
				bFlgLineScanOver:=FALSE;	
			END_IF*)
		
	        iAutoRunStep:=4070;	 

	ELSE  
       iAutoRunStep:=4080;	 
	END_IF
	
 ELSE   //IO线扫超240周期给结果      数据移位需要单独处理
	     IF  bFlgLineScanOver  THEN  //线扫超240周期给结果      数据移位需要单独处理
		
		 		FOR i1:=1 TO 20 BY 1 DO 																									
					IF i1<20 THEN
						 XianSaong_Up[20-i1]:=XianSaong_Up[19-i1];																						
					ELSE																				
						XianSaong_Up[0]:=CCD_COM.Scan.iResult_IO_UP;																											
					END_IF; 																							
				 END_FOR; 
				
				FOR i1:=1 TO 20 BY 1 DO 																									
					IF i1<20 THEN
						 XianSaong_Down[20-i1]:=XianSaong_Down[19-i1];																						
					ELSE																						
						XianSaong_Down[0]:=CCD_COM.Scan.iResult_IO_Down;																									
					END_IF; 																							
				 END_FOR;
		 	 
		 
			     IF XianSaong_Down[0]=30 AND XianSaong_Up[1]=30 THEN//---------------------------------线扫OK结果由8改为30，，，CCD需要同步更改
					   BeltData[BeltNo.NGBox1+2].fPoleNGSacnNo:=30; //线扫NG类型
				 ELSE
					//剔废前一工位汇总结果，5号位置，，，，，剔废工位为6
						IF XianSaong_Down[0]<>30 AND XianSaong_Up[1]=30 THEN
							BeltData[BeltNo.NGBox1+2].fPoleNGSacnNo:=XianSaong_Down[0];
						END_IF
		
						IF XianSaong_Down[0]=30 AND XianSaong_Up[1]<>30 THEN
							BeltData[BeltNo.NGBox1+2].fPoleNGSacnNo:=XianSaong_Up[1];
						END_IF
		
						IF XianSaong_Down[0]<>30 AND XianSaong_Up[1]<>30 THEN
							BeltData[BeltNo.NGBox1+2].fPoleNGSacnNo:=XianSaong_Up[1];
						END_IF			
				 END_IF	
				 
				 IF CCD_COM.Scan.iResult_IO_UP=33 AND NOT ProductPar.iModeEN.bCcdTcpEN AND NOT ProductPar.iModeEN.bLineScanCCDEN THEN
					stAlarm.arrFlowAlarm[25]:=TRUE;//上线扫超时报警
				END_IF	
				IF CCD_COM.Scan.iResult_IO_Down=33 AND NOT ProductPar.iModeEN.bCcdTcpEN AND NOT ProductPar.iModeEN.bLineScanCCDEN THEN
					stAlarm.arrFlowAlarm[27]:=TRUE;//下线扫超时报警
				END_IF	
			(*
           IF  CCD_COM.Scan.iResult_IO_UP<>33 AND CCD_COM.Scan.iResult_IO_Down<>33 THEN	
			     bFlgLineScanOver:=FALSE;	
		   END_IF*)
	 
	        iAutoRunStep:=4070;	 
	     ELSE  
             iAutoRunStep:=4080;	 
	    END_IF
 
 END_IF

 
 4070:
 	(*************************************************************************NG踢废********************************************************************************************)																										
	IF  (NOT ProductPar.iModeEN.bSizeCCDEN AND BeltData[BeltNo.NGBox1+2].fPoleNGSizeNo<>30  
		AND NOT ProductPar.iModeEN.bEmptyRunEN AND NOT ProductPar.iModeEN.bCcdTcpEN ) 		 
		OR			
	 	( BeltData[BeltNo.NGBox1+2].fPoleNGSacnNo <>30 AND NOT ProductPar.iModeEN.bCcdTcpEN AND NOT ProductPar.iModeEN.bLineScanCCDEN AND NOT ProductPar.iModeEN.bEmptyRunEN)  
		OR  
		(BeltData[BeltNo.NGBox1+2].bYellowMark)  OR 
	    (BeltData[BeltNo.NGBox1+2].bBlueMark)  THEN
		NG_Sum:=NG_Sum+1;
		arrCyCtrl[EvNo.	NGPushInsideAir	].Cmd.bON:=TRUE;//踢NG料打开
		arrCyCtrl[EvNo.	NGPushInsideAir	].Cmd.bOFF:=FALSE;//踢NG料关闭		
		arrCyCtrl[EVNo.NGPushInsideVacuo].Cmd.bON:=FALSE;//踢NG料真空打开
		arrCyCtrl[EVNo.NGPushInsideVacuo].Cmd.bOFF:=TRUE;//踢NG料真空关闭																	
		BeltData[BeltNo.NGBox1+2].bHavePole:=FALSE;	
		BeltData[BeltNo.NGBox1+2].stPoleNo:='';		
		nInt[3]:=1;																					
	ELSE	
		nInt[3]:=0;
		arrCyCtrl[EvNo.	NGPushInsideAir	].Cmd.bON:=FALSE;//踢NG料打开
		arrCyCtrl[EvNo.	NGPushInsideAir	].Cmd.bOFF:=TRUE;//踢NG料关闭		
		arrCyCtrl[EVNo.NGPushInsideVacuo].Cmd.bON:=TRUE;//踢NG料真空打开
		arrCyCtrl[EVNo.NGPushInsideVacuo].Cmd.bOFF:=FALSE;//踢NG料真空关闭																					
	END_IF	
	

    iAutoRunStep:=4080;	 
 
 
4080:


     Production.NGFlag[44]:=FALSE;//黄黄标跳切计数
	// Production.NGFlag[45]:=FALSE;//黄黄标计数
 	IF arrAxisCtrl[VirAxisNo.VirMain].Status.fModuloActPos>=310 THEN	
		bFlgLineScanOver:=FALSE;
	     CCD_COM.Scan.iResult_UP:=33; 
		 CCD_COM.Scan.iResult_Down:=33;	
	
		CCD_COM.Scan.iResult_IO_UP:=33;//复位线扫IO结果
		CCD_COM.Scan.iResult_IO_Down:=33;
		bLineScanResult1_UP:=FALSE;
		bLineScanResult2_UP:=FALSE;
		bLineScanResult1_Down:=FALSE;
		bLineScanResult2_Down:=FALSE;

		IF  NOT ProductPar.iModeEN.bCcdTcpEN AND NOT ProductPar.iModeEN.bLineScanCCDEN AND NOT ProductPar.iModeEN.bEmptyRunEN THEN
		    IF BeltData[BeltNo.NGBox1+2].fPoleNGSacnNo = 30 THEN
        	  iNGScane:=0;
			ELSE
              iNGScane:=iNGScane+1;
			END_IF  
		END_IF
													
		iAutoRunStep:=350;	
	END_IF	
 
																								
END_CASE	























(*
	//////////////////////模具前CCD检测计算极耳间距////////////////////////																								
			IF TabData[TabNo.MouldPhoto+1].bCCDed_M AND TabData[TabNo.MouldPhoto+2].bCCDed_M AND NOT TabData[TabNo.MouldPhoto+1].bTabOffsetNG_M AND NOT TabData[TabNo.MouldPhoto+2].bTabOffsetNG_M THEN																									
				fTabInteM_1:=PolePar.fPoleWidth+fDriverOffsetData[2]+(TabData[TabNo.MouldPhoto+2].fTab_OffsetM-TabData[TabNo.MouldPhoto+1].fTab_OffsetM);																								
			ELSE																									
				fTabInteM_1:=PolePar.fPoleWidth;																								
			END_IF																																																		
			InteData[InteNo.Mould-1].fTabIntervalM:=fTabInteM_1;																								
		
			IF TabData[TabNo.MouldPhoto+1].fPhotoPosM>TabData[TabNo.MouldPhoto+2].fPhotoPosM AND TabData[TabNo.MouldPhoto+1].bCCDed_M AND TabData[TabNo.MouldPhoto+2].bCCDed_M AND NOT TabData[TabNo.MouldPhoto+1].bTabOffsetNG_M AND NOT TabData[TabNo.MouldPhoto+2].bTabOffsetNG_M THEN																									
				fTabInteM_2:=TabData[TabNo.MouldPhoto+1].fPhotoPosM-TabData[TabNo.MouldPhoto+2].fPhotoPosM+(TabData[TabNo.MouldPhoto+2].fTab_OffsetM-TabData[TabNo.MouldPhoto+1].fTab_OffsetM);																								
			ELSE																									
				fTabInteM_2:=PolePar.fPoleWidth;																								
			END_IF																																																																						
		//////////////////////模具前极耳间距内前后肩宽状况判断////////////////////////	
			IF NOT ProductPar.iModeEN.bMouldXOffsetEN THEN																										
				IF ABS(InteData[InteNo.Mould-1].fTabIntervalM-PolePar.fPoleWidth)<=0.5 THEN//片宽偏差小于等于0.5																									
					InteData[InteNo.Mould-1].bTabInteFr_M:=FALSE;																								
					InteData[InteNo.Mould-1].bTabInteBe_M:=FALSE;																								
				ELSE																									
					IF NOT InteData[InteNo.Mould].bTabInteBe_M THEN																								
						InteData[InteNo.Mould-1].bTabInteFr_M:=FALSE;																							
						InteData[InteNo.Mould-1].bTabInteBe_M:=TRUE;																							
					ELSE																								
						InteData[InteNo.Mould-1].bTabInteFr_M:=TRUE;																							
						InteData[InteNo.Mould-1].bTabInteBe_M:=FALSE;																							
					END_IF																								
				END_IF		
			END_IF																							
		
			FOR i1:=1 TO 50 BY 1 DO 																									
					IF i1<50 THEN 																							
						 fM_TabInterData[51-i1]:=fM_TabInterData[50-i1];																																											
					ELSE																							
						fM_TabInterData[1]:=fTabInteM_1;																																											
					END_IF; 																							
			END_FOR; 

*)


(*																																														
//////////////////////蓝胶判断////////////////////////																										
	FOR i6:=1 TO 20 BY 1 DO																									
		IF fBluePos[21-i6]+PolePar.fBlue_Mould-PolePar.fPoleWidth<=TabData[TabNo.MouldPhoto+1].fPhotoPosM AND 																								
			fBluePos[21-i6]+PolePar.fBlue_Mould-PolePar.fPoleWidth>=TabData[TabNo.MouldPhoto+2].fPhotoPosM AND																							
			TabData[TabNo.MouldPhoto+1].fPhotoPosM>TabData[TabNo.MouldPhoto+2].fPhotoPosM AND																							
			TabData[TabNo.MouldPhoto+2].fPhotoPosM>0 AND																							
			fBluePos[21-i6]>0 THEN																							
			InteData[InteNo.Mould-1].bBlueNG:=TRUE;																							
			fBluePos[21-i6]:=0;																							
			EXIT;																							
		ELSE																								
			InteData[InteNo.Mould-1].bBlueNG:=FALSE;																							
		END_IF																								
	END_FOR		
*)			
(*																				
//////////////////////线扫判断////////////////////////																										
	FOR i7:=1 TO 20 BY 1 DO																									
		IF fLineScanPos[21-i7]+PolePar.fLineNG_Mould-PolePar.fPoleWidth<=TabData[TabNo.MouldPhoto+1].fPhotoPosM AND 																								
			fLineScanPos[21-i7]+PolePar.fLineNG_Mould-PolePar.fPoleWidth>=TabData[TabNo.MouldPhoto+2].fPhotoPosM AND																							
			TabData[TabNo.MouldPhoto+1].fPhotoPosM>TabData[TabNo.MouldPhoto+2].fPhotoPosM AND																							
			TabData[TabNo.MouldPhoto+2].fPhotoPosM>0 AND																							
			fLineScanPos[21-i7]>0 THEN																							
			InteData[InteNo.Mould-1].bLineScanNG:=TRUE;																							
			fLineScanPos[21-i7]:=0;																							
			EXIT;																							
		ELSE																								
			InteData[InteNo.Mould-1].bLineScanNG:=FALSE;																							
		END_IF																								
	END_FOR		
*)

   (*
//////////////裁切前黄标检测//////////
     FOR i1:=1 TO 10 BY 1 DO 																									
				IF i1<10 THEN 	
		           YellowmarkNG[11-i1]:=YellowmarkNG[10-i1];
				ELSE  
				   YellowmarkNG[1]:=1;
				END_IF;		
     END_FOR; 	
*)											

//裁断后数据移位													
///////////////////////首位给记忆/////////////////////////		
(*																																																
	IF arrAxisCtrl[AxisNo.Cuter].Status.NoMoving OR fbCuterCam.iTableSel<>1 THEN																									
		iNormalCuter:=0;																								
		bJumpCut:=TRUE;																								
	ELSE																									
		iNormalCuter:=iNormalCuter+1;																								
	END_IF																									
	IF NOT bJumpCut THEN																									
		BeltData[1].iJumpCutNG:=1;//判断切刀NoMoving+1个周期，给2																								
	ELSE																									
		BeltData[1].iJumpCutNG:=2;																								
	END_IF			
*)



(*																								
	IF (InteData[InteNo.Cuter-1].bBlueNG AND NOT ProductPar.iModeEN.bFlgBlueEN OR InteData[InteNo.Cuter-1].bLineScanNG AND NOT ProductPar.iModeEN.bLineScanCCDEN) AND NOT ProductPar.iModeEN.bEmptyRunEN THEN																									
		IF iCuterRunTableSel=1 THEN																								
			fbCuterCam.iTableSel:=2;																							
		ELSE																								
			fbCuterCam.iTableSel:=3; 																							
		END_IF;//裁切凸轮切换为stop																								
	ELSE																									
		fbCuterCam.iTableSel:=1;//裁切凸轮切换为正常																								
	END_IF		
*)		


(*
///////////////////////监测皮带上的记忆/////////////////////////																				
	iBeltNoPeaceCount:=0;																									
	bPeaceBelt1Front:=FALSE;																									
	FOR i1:=1 TO BeltNo.SubBelt1 BY 1 DO 																									
		   bPeaceBelt1Front:=bPeaceBelt1Front OR BeltData[i1].bHavePole ;																								
		   IF iPoleCarryEver=1 AND NOT BeltData[i1].bHavePole THEN																								
			   iBeltNoPeaceCount:=iBeltNoPeaceCount+1;																							
		   END_IF		   																						
	END_FOR;																									
	bPeaceBelt2Front:=FALSE;																									
	FOR i1:=1 TO BeltNo.SubBelt2 BY 1 DO 																									
		   bPeaceBelt2Front:=bPeaceBelt2Front OR BeltData[i1].bHavePole ;																								
		   IF iPoleCarryEver=2 AND NOT BeltData[i1].bHavePole THEN																								
			   iBeltNoPeaceCount:=iBeltNoPeaceCount+1;																							
		   END_IF																								
	END_FOR;																									
	bPeaceBelt3Front:=FALSE;																									
																										
	FOR i1:=1 TO BeltNo.SubBelt3 BY 1 DO 																									
		   bPeaceBelt3Front:=bPeaceBelt3Front OR BeltData[i1].bHavePole ;																								
		   IF iPoleCarryEver=3 AND NOT BeltData[i1].bHavePole THEN																								
			   iBeltNoPeaceCount:=iBeltNoPeaceCount+1;																							
		   END_IF																								
	END_FOR;																									
		bHavePeaceBelt:=FALSE;																								
	FOR i1:=1 TO BeltNo.SubBelt2 BY 1 DO 																									
		   bPeaceBelt2Front:=bPeaceBelt2Front OR BeltData[i1].bHavePole ;																								
	END_FOR;		
*)
END_ACTION

ACTION F0505MainAuto5:

///////////////////////////////////////////////////主轴运行中，主驱&皮带停止，主轴当前周期即将结束。判断皮带耦合状况，主轴运行模式判断 //////////////////////////////////////////////////////////
CASE iAutoRunStep OF 
	
5000://皮带耦合请求
    
   IF  bBelt1Taking  THEN	 ////////////////////////
	   		iMainMode:=1;	
			bBelt1Gearask:=TRUE;
			bBelt2Gearask:=FALSE;
			bBelt3Gearask:=FALSE;
			iStopCount2:=iStopCount2+1;
			iAutoRunStep:=5015;	
   ELSIF  bBelt2Taking  THEN		   /////////////////
		
		   IF NOT bBelt1Taking  THEN   // 1# 2#  
				IF  NOT	 BeltData[BeltNo.SubBelt1].bHavePole  THEN
					 bBelt1Gearask:=TRUE;
					 bBelt2Gearask:=FALSE;
					 bBelt3Gearask:=FALSE;	
					iMainMode:=2;	
					iAutoRunStep:=5015;	
			    ELSE
					iMainMode:=1;	
					bBelt1Gearask:=TRUE;
					bBelt2Gearask:=FALSE;
					bBelt3Gearask:=FALSE;
					iAutoRunStep:=5015;	
			    END_IF	
		   ELSE
				iMainMode:=1;	
				bBelt1Gearask:=TRUE;
				bBelt2Gearask:=FALSE;
				bBelt3Gearask:=FALSE;
				iAutoRunStep:=5015;	
           END_IF 	 
		   
		   
    ELSIF bBelt3Taking  THEN     //3# 取片中 //////////////////////
		
		 IF NOT BeltData[BeltNo.SubBelt1].bHavePole THEN//分段1运行							
			bBelt1Gearask:=TRUE;
			bBelt2Gearask:=FALSE;
			bBelt3Gearask:=FALSE;
			iMainMode:=2;						
		ELSIF BeltData[BeltNo.SubBelt1].bHavePole AND //	bBelt2Need AND 									
			NOT BeltData[BeltNo.SubBelt2].bHavePole THEN 	//分段1/2运行										
			bBelt1Gearask:=TRUE;
			bBelt2Gearask:=TRUE;
			bBelt3Gearask:=FALSE;	
			iMainMode:=2;	
        ELSIF BeltData[BeltNo.SubBelt1].bHavePole AND BeltData[BeltNo.SubBelt2].bHavePole  THEN   
         	bBelt1Gearask:=TRUE;
			bBelt2Gearask:=FALSE;
			bBelt3Gearask:=FALSE;	
			iMainMode:=1; 													
		END_IF	
		iAutoRunStep:=5015;	
				
   ELSE
	
		IF 	NOT BeltData[BeltNo.SubBelt1].bHavePole THEN//分段1运行							
			bBelt1Gearask:=TRUE;
			bBelt2Gearask:=FALSE;
			bBelt3Gearask:=FALSE;	
			 iMainMode:=2;					
		ELSIF BeltData[BeltNo.SubBelt1].bHavePole AND 	//bBelt2Need AND 									
			NOT BeltData[BeltNo.SubBelt2].bHavePole THEN 	//分段1/2运行										
			bBelt1Gearask:=TRUE;
			bBelt2Gearask:=TRUE;
			bBelt3Gearask:=FALSE;	
			 iMainMode:=2;														
		ELSIF bBelt2Need AND bBelt3Need AND 
			BeltData[BeltNo.SubBelt1].bHavePole AND 										
			BeltData[BeltNo.SubBelt2].bHavePole  AND    (   NOT BeltData[BeltNo.SubBelt3].bHavePole OR (BeltData[BeltNo.SubBelt3].bHavePole AND BeltData[BeltNo.SubBelt3].stPoleNo=''AND NOT ProductPar.iModeEN.bCcdTcpEN AND NOT ProductPar.iModeEN.bSizeCCDEN)   OR     ProductPar.iModeEN.bP2PartEN    )    THEN 	//分段1/2/3运行									
			bBelt1Gearask:=TRUE;
			bBelt2Gearask:=TRUE;
			bBelt3Gearask:=TRUE; 
			 iMainMode:=2;	
        ELSIF   BeltData[BeltNo.SubBelt1].bHavePole  AND   BeltData[BeltNo.SubBelt2].bHavePole   AND  BeltData[BeltNo.SubBelt3].bHavePole AND BeltData[BeltNo.SubBelt3].stPoleNo<>'' AND NOT ProductPar.iModeEN.bP2PartEN   THEN
              iMainMode:=1;	
			  bBelt1Gearask:=TRUE;
			  bBelt2Gearask:=FALSE;
			  bBelt3Gearask:=FALSE;													
		END_IF	
		 iAutoRunStep:=5015;	   
END_IF

5015:
	IF bBelt1Gearask AND NOT bBelt2Gearask AND NOT bBelt3Gearask THEN//分段1运行	
		bSubBelt2fratio:=FALSE;
		bSubBelt3fratio:=FALSE;															
	ELSIF bBelt1Gearask AND bBelt2Gearask AND NOT bBelt3Gearask THEN //分段1/2运行		
		bSubBelt2fratio:=TRUE;
		bSubBelt3fratio:=FALSE;																			
	ELSIF bBelt1Gearask AND bBelt2Gearask AND bBelt3Gearask THEN //分段1/2/3运行		
		bSubBelt2fratio:=TRUE;
		bSubBelt3fratio:=TRUE;				
	END_IF	
	iAutoRunStep:=5020;	

	
5020:	
    	IF   bBelt1Taking  THEN
		iAutoAuxStep6Temp:=iAutoAuxStep6;     //记录超周期时候步序
		iOverCycleCount1:=iOverCycleCount1+1;//超周期计数
	END_IF
	 IF   bBelt2Taking  THEN
		   iAutoAuxStep7Temp:=iAutoAuxStep7;    //记录超周期时候步序
		   iOverCycleCount2:=iOverCycleCount2+1;//超周期计数
	 END_IF 
	 IF   bBelt3Taking  THEN
		  iAutoAuxStep8Temp:=iAutoAuxStep8;    //记录超周期时候步序
		  iOverCycleCount3:=iOverCycleCount3+1;//超周期计数
	 END_IF 
	
	(*
	  IF iMainMode=2 THEN 
		 IF  NOT bBelt1Taking  THEN
			iAutoAuxStep6:=0;
			InterPart.M1Allow:=FALSE;
		 END_IF
		 IF  NOT bBelt2Taking	AND NOT BeltData[BeltNo.SubBelt3].bHavePole  THEN
			iAutoAuxStep7:=0;
			InterPart.M2Allow:=FALSE;
		 END_IF 
		 //IF  NOT bBelt3Taking  THEN
				//iAutoAuxStep8:=0;
				//InterPart.M3Allow:=FALSE;
		 //END_IF
	  END_IF  *)  
	  
	  IF  itest=3 AND  iMainMode=1 THEN
		  iMainMode:=3;
		  iStopCount3:=iStopCount3+1;
		  stAlarm.arrLightWarn[11]:=TRUE; 
	  END_IF
	  
	  
	  IF bMA21 AND  itest=3 AND  iMainMode=2 THEN
	      iMainMode:=3;
	      stAlarm.arrLightWarn[11]:=TRUE; 
		  bMA21:=FALSE;
	  END_IF
	 
	iPoleNoHave1:=iPoleNoHaveA;
	iAutoRunStep:=5030;	
	
	
5030://判断运行模式
	IF stSysState.Stoping THEN
		(*
		IF NOT bFlgStoping THEN
			IF iMainMode=1 OR stSysState.btnEstop THEN
				iAutoRunStep:=500;//异常情况,主轴当前周期立即停止
				bSysStoping:=TRUE;
			ELSE
				iAutoRunStep:=400;//再走一个周期
				bSysStoping:=TRUE;					
			END_IF
		ELSE
			iAutoRunStep:=450;//等待主轴停止
			bSysStoping:=TRUE;
		END_IF *)
		
	   IF NOT bFlgStoping THEN
			IF iMainMode=1  THEN
				bSysStoping:=TRUE;
				iAutoRunStep:=450;
				itest2:=1;
			ELSIF iMainMode=2 THEN
				iAutoRunStep:=400;//再走一个周期
				bSysStoping:=TRUE;
                itest2:=2;	
			ELSIF iMainMode=3 THEN
				iAutoRunStep:=500;//
				bSysStoping:=TRUE;	
                itest2:=3;				
			END_IF
		ELSE
			iAutoRunStep:=450;//等待主轴停止
			bSysStoping:=TRUE;
			 itest2:=4;	 
		END_IF
	END_IF	
	
	
	
  IF NOT stSysState.Stoping THEN
		IF iMainMode=1 THEN
			IF NOT bFlgStoping THEN
				//iAutoRunStep:=500;//异常情况,主轴当前周期立即停止
				iAutoRunStep:=450;
				//itest1:=1;
				//itest2:=iPoleNoHave1;	
			   iStopCount:=iStopCount+1;
			    itest2:=11;	
			ELSE
				iStopCount:=iStopCount+1;
				iAutoRunStep:=450;//等待主轴停止
				  itest2:=12;	
			END_IF
			
		ELSIF iMainMode=2 THEN
			IF iPoleNoHave1=1 THEN
				iAutoRunStep:=400;//再走一个周期
				  itest2:=13;	
			ELSIF iPoleNoHave1=2 THEN
				bFlgStoping:=FALSE;
				arrAxisCtrl[VirAxisNo.VirMain].Cmd.bMoveVelo:=FALSE;
				iAutoRunStep:=150;//再走多个周期	
				  itest2:=14;	
			ELSIF iPoleNoHave1=0 THEN
				IF NOT bFlgStoping THEN
					//iAutoRunStep:=500;//异常情况,主轴当前周期立即停止   400
					iAutoRunStep:=450;
					itest1:=itest1+1;
					  itest2:=15;	
					//itest2:=iPoleNoHave1;
					//itest3:=iPoleNoHaveA;
				ELSE
					//itest2:=itest2+1;
					iAutoRunStep:=450;//等待主轴停止
					  itest2:=16;	
				END_IF
			END_IF	
        ELSIF iMainMode=3 THEN
		   iAutoRunStep:=500;//异常情况,主轴当前周期立即停止
		     itest2:=17;	
		END_IF
  END_IF
	
	//bBelt1Gearask:=FALSE;
	bBelt2Gearask:=FALSE;
	bBelt3Gearask:=FALSE;		
END_CASE







(*
	
5030://判断运行模式
	IF stSysState.Stoping THEN
		IF NOT bFlgStoping THEN
			IF iMainMode=1 OR stSysState.btnEstop THEN
				iAutoRunStep:=500;//异常情况,主轴当前周期立即停止
				bSysStoping:=TRUE;
			ELSE
				iAutoRunStep:=400;//再走一个周期
				bSysStoping:=TRUE;					
			END_IF
		ELSE
			iAutoRunStep:=450;//等待主轴停止
			bSysStoping:=TRUE;
		END_IF
	END_IF	
	
	IF NOT stSysState.Stoping THEN
		IF iMainMode=1 THEN
			IF NOT bFlgStoping THEN
				//iAutoRunStep:=500;//异常情况,主轴当前周期立即停止
				iAutoRunStep:=400;
				itest1:=1;
				itest2:=iPoleNoHave1;	
			   iStopCount:=iStopCount+1;
			ELSE
				iAutoRunStep:=450;//等待主轴停止
			END_IF
		ELSIF iMainMode=2 THEN
			IF iPoleNoHave1=1 THEN
				iAutoRunStep:=400;//再走一个周期
			ELSIF iPoleNoHave1=2 THEN
				bFlgStoping:=FALSE;
				arrAxisCtrl[VirAxisNo.VirMain].Cmd.bMoveVelo:=FALSE;
				iAutoRunStep:=150;//再走多个周期	
			ELSIF iPoleNoHave1=0 THEN
				IF NOT bFlgStoping THEN
					//iAutoRunStep:=500;//异常情况,主轴当前周期立即停止   400
					iAutoRunStep:=400;
					itest1:=2;
					itest2:=iPoleNoHave1;
					itest3:=iPoleNoHaveA;
				ELSE
					iAutoRunStep:=450;//等待主轴停止
				END_IF
			END_IF			
		END_IF
	 END_IF
	
	bBelt1Gearask:=FALSE;
	bBelt2Gearask:=FALSE;
	bBelt3Gearask:=FALSE;		
*)















(*
5000://皮带耦合请求
   IF   ( InterPart.M1Allow  OR  bBelt1Taking )  OR         //没取玩后者  锁定取片中
           ( InterPart.M2Allow  OR  bBelt2Taking )  OR     //没取玩后者  锁定取片中
            (InterPart.M3Allow  OR  bBelt3Taking )     THEN    //没取玩后者  锁定取片中  THEN
			 	bSubBelt2fratio:=FALSE;
				bSubBelt3fratio:=FALSE;	
            	iMainMode:=1;		
                iAutoRunStep:=5015;	
    ELSE	
		
			IF 	NOT BeltData[BeltNo.SubBelt1].bHavePole THEN//分段1运行							
				bBelt1Gearask:=TRUE;
				bBelt2Gearask:=FALSE;
				bBelt3Gearask:=FALSE;									
			ELSIF bBelt2Need AND BeltData[BeltNo.SubBelt1].bHavePole AND 										
					 NOT BeltData[BeltNo.SubBelt2].bHavePole THEN 	//分段1/2运行										
				bBelt1Gearask:=TRUE;
				bBelt2Gearask:=TRUE;
				bBelt3Gearask:=FALSE;																		
			ELSIF bBelt2Need AND bBelt3Need AND 
					 BeltData[BeltNo.SubBelt1].bHavePole AND 										
					 BeltData[BeltNo.SubBelt2].bHavePole  AND    (   NOT BeltData[BeltNo.SubBelt3].bHavePole   OR     ProductPar.iModeEN.bP2PartEN    )    THEN 	//分段1/2/3运行									
				bBelt1Gearask:=TRUE;
				bBelt2Gearask:=TRUE;
				bBelt3Gearask:=TRUE;																		
			END_IF	
		 iMainMode:=2;	
	     iAutoRunStep:=5010;
		 
  END_IF

*)


(*

5010:
	IF 	NOT BeltData[BeltNo.SubBelt1].bHavePole THEN//分段1运行							
		bBelt1Gearask:=TRUE;
		bBelt2Gearask:=FALSE;
		bBelt3Gearask:=FALSE;									
	ELSIF bBelt2Need AND BeltData[BeltNo.SubBelt1].bHavePole AND 										
		NOT BeltData[BeltNo.SubBelt2].bHavePole THEN 	//分段1/2运行										
		bBelt1Gearask:=TRUE;
		bBelt2Gearask:=TRUE;
		bBelt3Gearask:=FALSE;																					
	END_IF	
	iAutoRunStep:=5015;	

	
5011://综合判断皮带耦合
	IF 	NOT BeltData[BeltNo.SubBelt1].bHavePole THEN//分段1运行							
		bBelt1Gearask:=TRUE;
		bBelt2Gearask:=FALSE;
		bBelt3Gearask:=FALSE;									
	ELSIF bBelt2Need AND BeltData[BeltNo.SubBelt1].bHavePole AND 										
		NOT BeltData[BeltNo.SubBelt2].bHavePole THEN 	//分段1/2运行										
		bBelt1Gearask:=TRUE;
		bBelt2Gearask:=TRUE;
		bBelt3Gearask:=FALSE;																		
	ELSIF bBelt2Need AND bBelt3Need AND 
		BeltData[BeltNo.SubBelt1].bHavePole AND 										
		BeltData[BeltNo.SubBelt2].bHavePole  AND    (   NOT BeltData[BeltNo.SubBelt3].bHavePole   OR     ProductPar.iModeEN.bP2PartEN    )    THEN 	//分段1/2/3运行									
		bBelt1Gearask:=TRUE;
		bBelt2Gearask:=TRUE;
		bBelt3Gearask:=TRUE;																		
	END_IF	
	iAutoRunStep:=5015;		

*)









(*
	
5010://综合判断皮带耦合
//IF arrAxisCtrl[VirAxisNo.VirMain].Status.fModuloActPos>=345 AND arrAxisCtrl[VirAxisNo.VirMain].Status.fModuloActPos<355 THEN//345   355
	IF bBelt1Gearask AND NOT bBelt2Gearask AND NOT bBelt3Gearask THEN//分段1运行	
		IF NOT bBelt1Taking THEN
			bSubBelt2fratio:=FALSE;
			bSubBelt3fratio:=FALSE;														
			iMainMode:=2;
		ELSE	
			bSubBelt2fratio:=FALSE;
			bSubBelt3fratio:=FALSE;											
			iMainMode:=1;		
		 END_IF			
	ELSIF bBelt1Gearask AND bBelt2Gearask AND NOT bBelt3Gearask THEN //分段1/2运行		
			IF NOT bBelt1Taking  AND NOT   bBelt2Taking  THEN
				bSubBelt2fratio:=TRUE;
				bSubBelt3fratio:=FALSE;																			
				iMainMode:=2;				
			ELSE
				bSubBelt2fratio:=FALSE;
				bSubBelt3fratio:=FALSE;											
				iMainMode:=1;								
			END_IF	
	ELSIF bBelt1Gearask AND bBelt2Gearask AND bBelt3Gearask THEN //分段1/2/3运行		
			IF NOT bBelt1Taking AND NOT bBelt2Taking  AND NOT bBelt3Taking    THEN
				bSubBelt2fratio:=TRUE;
				bSubBelt3fratio:=TRUE;		
				iMainMode:=2;														
			ELSE
				bSubBelt2fratio:=FALSE;
				bSubBelt3fratio:=FALSE;												
				iMainMode:=1;							
			END_IF						
	END_IF
		iAutoRunStep:=5015;
//END_IF

5015:	
	(************************下个周期皮带启动异常报警************************)
		    IF   bBelt1Taking  THEN
				   iAutoAuxStep6Temp:=iAutoAuxStep6;     //记录超周期时候步序
				   iOverCycleCount1:=iOverCycleCount1+1;//超周期计数
			 END_IF
			  IF   bBelt2Taking  THEN
				   iAutoAuxStep7Temp:=iAutoAuxStep7;    //记录超周期时候步序
				   iOverCycleCount2:=iOverCycleCount2+1;//超周期计数
			 END_IF 
			 IF   bBelt3Taking  THEN
					  iAutoAuxStep8Temp:=iAutoAuxStep8;    //记录超周期时候步序
					  iOverCycleCount3:=iOverCycleCount3+1;//超周期计数
			 END_IF 
	
	  IF iMainMode=2 THEN 
			  IF  NOT bBelt1Taking  THEN
					iAutoAuxStep6:=0;
					InterPart.M1Allow:=FALSE;
			 END_IF
			  IF  NOT bBelt2Taking	AND NOT BeltData[BeltNo.SubBelt3].bHavePole  THEN
					iAutoAuxStep7:=0;
					InterPart.M2Allow:=FALSE;
			 END_IF 
			 //IF  NOT bBelt3Taking  THEN
					//iAutoAuxStep8:=0;
					//InterPart.M3Allow:=FALSE;
			 //END_IF
	  END_IF
	 
	iPoleNoHave1:=iPoleNoHaveA;
	iAutoRunStep:=5020;

5020://判断运行模式
	IF stSysState.Stoping THEN
		IF NOT bFlgStoping THEN
			IF iMainMode=1 OR stSysState.btnEstop THEN
				iAutoRunStep:=500;//异常情况,主轴当前周期立即停止
				bSysStoping:=TRUE;
			ELSE
				iAutoRunStep:=400;//再走一个周期
				bSysStoping:=TRUE;					
			END_IF
		ELSE
			iAutoRunStep:=450;//等待主轴停止
			bSysStoping:=TRUE;
		END_IF
	ELSE
		IF iMainMode=1 THEN
			IF NOT bFlgStoping THEN
				iAutoRunStep:=500;//异常情况,主轴当前周期立即停止
				itest1:=1;
				itest2:=iPoleNoHave1;
				bTest[11]:=bBelt1Gearask;
				bTest[12]:=bBelt2Gearask;
				bTest[13]:=bBelt3Gearask;
				bTest[14]:=bBelt1Taking;
				bTest[15]:=bBelt2Taking;		
               iStopCount:=iStopCount+1;
			ELSE
				iAutoRunStep:=450;//等待主轴停止
			END_IF
		ELSE
			IF iPoleNoHave1=1 THEN
				iAutoRunStep:=400;//再走一个周期
			ELSIF iPoleNoHave1=2 THEN
				bFlgStoping:=FALSE;
				iAutoRunStep:=150;//再走多个周期	
				(*
				IF arrAxisCtrl[VirAxisNo.VirMain].Status.Moving THEN
					iAutoRunStep:=150;//再走多个周期
				ELSE
					arrAxisPar[VirAxisNo.VirMain].fVelocity_of_Velo:=PolePar.iMainVel*6;
					arrAxisCtrl[VirAxisNo.VirMain].Cmd.bMoveVelo:=TRUE;
				END_IF	
				*)
			ELSIF iPoleNoHave1=0 THEN
				
				IF NOT bFlgStoping THEN
					iAutoRunStep:=400;//异常情况,主轴当前周期立即停止
					itest1:=2;
					itest2:=iPoleNoHave1;
					itest3:=iPoleNoHaveA;
					bTest[11]:=bBelt1Gearask;
					bTest[12]:=bBelt2Gearask;
					bTest[13]:=bBelt3Gearask;
					bTest[14]:=bBelt1Taking;
					bTest[15]:=bBelt2Taking;
				ELSE
					iAutoRunStep:=450;//等待主轴停止
				END_IF
			END_IF			
		END_IF
	END_IF
	bBelt1Gearask:=FALSE;
	bBelt2Gearask:=FALSE;
	bBelt3Gearask:=FALSE;			

*)
END_ACTION

ACTION F0506MainAuto6:
//////////////////////////////////////////////主轴静止中，由于皮带料满，主轴运动自动停止,判断皮带耦合状况. 继续与叠片交互//////////////////////////////////////////////////////

DelayStep6(IN:= , PT:=T#2MS , Q=> , ET=> );
CASE iAutoRunStep OF 
6000://
	IF iPoleNoHaveA=0 THEN
		iAutoRunStep:=6010;//皮带上料全满
	ELSIF    NOT bBelt1Taking  AND  NOT  InterPart.M1Allow   AND  
                NOT bBelt2Taking  AND  NOT  InterPart.M2Allow   AND 
                NOT bBelt3Taking  AND  NOT  InterPart.M3Allow   THEN
		iAutoAuxStep6:=0;
		InterPart.M1Allow:=FALSE;	
		iAutoAuxStep7:=0;
		InterPart.M2Allow:=FALSE;				
		iAutoAuxStep8:=0;
		InterPart.M3Allow:=FALSE;
		iAutoRunStep:=100;//皮带上料未满,返回继续切片送料
	END_IF	
6010://
	IF (iPoleCarryEver=3 AND 
        (NOT bBelt1Taking AND  NOT  InterPart.M1Allow  AND 
         NOT bBelt2Taking AND  NOT  InterPart.M2Allow  AND
         NOT bBelt3Taking AND  NOT  InterPart.M3Allow     )      ) OR
	
		(iPoleCarryEver=2 AND (NOT bBelt1Taking AND NOT bBelt2Taking )) OR
		(iPoleCarryEver=1 AND NOT bBelt1Taking )  THEN
		iAutoRunStep:=6020;//
	ELSE
		iAutoRunStep:=6000;//
	END_IF
	
6020://
	IF iPoleCarryEver=3 THEN
		IF BeltData[BeltNo.SubBelt1].bHavePole //AND ((*BeltData[BeltNo.SubBelt1].stPoleNo<>'' OR*) ProductPar.iModeEN.bCcdTcpEN)
			AND BeltData[BeltNo.SubBelt2].bHavePole //AND ((*BeltData[BeltNo.SubBelt2].stPoleNo<>'' OR*) ProductPar.iModeEN.bCcdTcpEN)
			AND BeltData[BeltNo.SubBelt3].bHavePole //AND ((*BeltData[BeltNo.SubBelt3].stPoleNo<>'' OR*) ProductPar.iModeEN.bCcdTcpEN)
			AND (iAutoAuxStep9=0 OR iAutoAuxStep9=666)  THEN
			iAutoAuxStep9:=100;
		END_IF			
	ELSIF iPoleCarryEver=2 THEN
		IF BeltData[BeltNo.SubBelt1].bHavePole AND (BeltData[BeltNo.SubBelt1].stPoleNo<>''OR ProductPar.iModeEN.bCcdTcpEN)
			AND BeltData[BeltNo.SubBelt2].bHavePole AND (BeltData[BeltNo.SubBelt2].stPoleNo<>''OR ProductPar.iModeEN.bCcdTcpEN)
			AND    NOT  bBelt1Taking AND   iAutoAuxStep6<>20     THEN
			iAutoAuxStep6:=10;
			//bBelt1Taking:=TRUE;
		END_IF
		IF BeltData[BeltNo.SubBelt2].bHavePole  AND  (BeltData[BeltNo.SubBelt2].stPoleNo<>''OR ProductPar.iModeEN.bCcdTcpEN)
			AND NOT  bBelt2Taking AND   iAutoAuxStep7<>20  THEN
			iAutoAuxStep7:=10;
			//bBelt2Taking:=TRUE;
		END_IF
	ELSE
		IF BeltData[BeltNo.SubBelt1].bHavePole AND (BeltData[BeltNo.SubBelt1].stPoleNo<>'' OR ProductPar.iModeEN.bCcdTcpEN OR ProductPar.iModeEN.bSizeCCDEN)
		AND  NOT  bBelt1Taking AND   iAutoAuxStep6<>20        THEN
			iAutoAuxStep6:=10;
			//bBelt1Taking:=TRUE;
		END_IF	
	END_IF	
	DelayStep6.IN:=TRUE;
	iAutoRunStep:=6030;		
(*	
6020://
		IF iPoleCarryEver=3 THEN
			IF BeltData[BeltNo.SubBelt1].bHavePole AND BeltData[BeltNo.SubBelt2].bHavePole AND BeltData[BeltNo.SubBelt3].bHavePole  THEN	
					IF (InterPart.M1LockReady OR InterPart.M1JumpReady) AND (InterPart.M2LockReady OR InterPart.M2JumpReady) AND
					   (InterPart.M3LockReady OR InterPart.M3JumpReady) THEN
							IF 	InterPart.M1LockReady AND NOT bBelt1Taking AND NOT  InterPart.M1Allow  THEN
								iAutoAuxStep6:=10;
							END_IF
							IF 	InterPart.M2LockReady AND NOT bBelt2Taking AND NOT  InterPart.M2Allow   THEN
								iAutoAuxStep7:=10;
							END_IF	
							IF 	InterPart.M3LockReady AND NOT bBelt3Taking AND NOT  InterPart.M3Allow   THEN
								iAutoAuxStep8:=10;
							END_IF		
					END_IF		
			END_IF			

	
		ELSIF iPoleCarryEver=2 THEN
			IF BeltData[BeltNo.SubBelt1].bHavePole AND BeltData[BeltNo.SubBelt2].bHavePole AND    NOT  bBelt1Taking AND   iAutoAuxStep6<>20     THEN
				iAutoAuxStep6:=10;
				//bBelt1Taking:=TRUE;
			END_IF
			IF BeltData[BeltNo.SubBelt2].bHavePole  AND    NOT  bBelt2Taking AND   iAutoAuxStep7<>20  THEN
				iAutoAuxStep7:=10;
				//bBelt2Taking:=TRUE;
			END_IF
		ELSE
			IF BeltData[BeltNo.SubBelt1].bHavePole  AND  NOT  bBelt1Taking AND   iAutoAuxStep6<>20        THEN
				iAutoAuxStep6:=10;
				//bBelt1Taking:=TRUE;
			END_IF	
		END_IF
		
		DelayStep6.IN:=TRUE;
		iAutoRunStep:=6030;
*)
6030:		
		IF DelayStep6.Q THEN
			DelayStep6.IN:=FALSE;
			iAutoRunStep:=6000;
		END_IF
				
END_CASE
END_ACTION

ACTION F0511CCDAuto:


///////////////////////////////////////////////////////////尺寸检测///////////////////////////////////////////////////////////////////
CASE iAutoAuxStep3 OF
10://
	IF arrAxisCtrl[VirAxisNo.VirMain].Status.fActPos < fRecordOverHangInMainPos-fRecordOverHangInMainPosMod+360+ProductPar.parPublic.fMainPos-10 THEN//到下个周期250度以前有效
		IF arrAxisCtrl[VirAxisNo.VirMain].Status.fActPos>=fRecordOverHangInMainPos+30 THEN
			IF CCD_COM.Size.iFinish=1 OR CCD_COM.Size.iFinish=2 OR CCD_COM.Size.iFinish=3 THEN
					IF 1<=CCD_COM.Size.fPoleNGSizeNo AND CCD_COM.Size.fPoleNGSizeNo<=30 THEN
						BeltData[BeltNo.OverHang].fPoleHeigh:=CCD_COM.Size.fPoleHeigh;//极片高；
						BeltData[BeltNo.OverHang].fPoleWidth:=CCD_COM.Size.fPoleWidth;//极片长（运行方向）；
						BeltData[BeltNo.OverHang].stPoleNo:=CCD_COM.Size.stPoleNo;//
						
						BeltData[BeltNo.OverHang].fTabWidth:=CCD_COM.Size.fTabWidth;  //尺寸检测CCD结果(极耳宽度)
						BeltData[BeltNo.OverHang].fTabHeigh:=CCD_COM.Size.fTabHeigh;  //尺寸检测CCD结果(极耳高度)
						BeltData[BeltNo.OverHang].fTabSite:=CCD_COM.Size.fTabSite; // 极耳左，右边距(就是极耳位置，不分左右)
						//BeltData[BeltNo.OverHang].fOffsetDeg:=CCD_COM.Size.fOffsetDeg; //尺寸检测CCD结果(极片裁切面角度偏移)
						
						BeltData[BeltNo.OverHang].RoundedSize1:=CCD_COM.Size.RoundedSize1   ;//        圆角尺寸1 面积   叠片侧(正极)       负极相反
						BeltData[BeltNo.OverHang].RoundedSize2:=CCD_COM.Size.RoundedSize2   ;//        圆角尺寸2 面积    切刀侧(正极)        负极相反
						BeltData[BeltNo.OverHang].RoundedSize3:=CCD_COM.Size.RoundedSize3  ;//        圆角尺寸3纵深 叠片侧(正极)        负极相反
						BeltData[BeltNo.OverHang].RoundedSize4:=CCD_COM.Size.RoundedSize4   ;//        圆角尺寸4纵深 切刀侧(正极)     负极相反
						BeltData[BeltNo.OverHang].RoundedSize5:=CCD_COM.Size.RoundedSize5   ;//        圆角尺寸5 横深
						BeltData[BeltNo.OverHang].RoundedSize6:=CCD_COM.Size.RoundedSize6  ;//        圆角尺寸6横深
						BeltData[BeltNo.OverHang].RoundedSize7:=CCD_COM.Size.RoundedSize7   ;//        圆角尺寸7横深 叠片侧(正极)     负极相反
						BeltData[BeltNo.OverHang].RoundedSize8:=CCD_COM.Size.RoundedSize8  ;//        圆角尺寸8横深 切刀侧(正极)     负极相反
						
						BeltData[BeltNo.OverHang].PolePlateAngle1 :=CCD_COM.Size.PolePlateAngle1 ;//        极片角度1  极片角度
						BeltData[BeltNo.OverHang].PolePlateAngle2:=CCD_COM.Size.PolePlateAngle2  ;//        极片角度2
						BeltData[BeltNo.OverHang].PolePlateAngle3:=CCD_COM.Size.PolePlateAngle3   ;//        极片角度3
						BeltData[BeltNo.OverHang].PolePlateAngle4:=CCD_COM.Size.PolePlateAngle4   ;//        极片角度4
						BeltData[BeltNo.OverHang].fPoleNGSizeNo:=CCD_COM.Size.fPoleNGSizeNo;  //尺寸检测CCD结果(NG分类编号)
						BeltData[BeltNo.OverHang].iPoleRAngleNG:=CCD_COM.Size.iPoleRAngleNG;//尺寸检测CCD结果(R角NG)
						BeltData[BeltNo.OverHang].iFinish:=CCD_COM.Size.iFinish;  //尺寸检测CCD结果指示(1=完成;2=NG;3=无片;0=无效)  SizeResults
						BeltData[BeltNo.OverHang].AppearanceResult:=CCD_COM.Size.AppearanceResult;// 极片外观判定结果   线扫NG、OK
						BeltData[BeltNo.OverHang].PolePlateLenth :=CCD_COM.Size.fTabWidth ;// 极片外观判定结果   线扫NG、OK
						//BeltData[BeltNo.OverHang].SlicingSpeed:=GVL_Par.ProductPar.AnPar.iMainVel;//切片速度PPM;
						//BeltData[BeltNo.OverHang].UnreelingTension :=ABS(GMotion.iTargetTorque[1]);//放卷张力  %；
						BeltData[BeltNo.OverHang].SlicingSpeed:=PolePar.fSpeed;//切片速度PPM;
						//BeltData[BeltNo.OverHang].UnreelingTension :=(480+ab);
						CCD_Rounde.CCD_Enable:=TRUE;//R纠偏闭环数据记录开始
						
						//BeltData[BeltNo.OverHang].UnreelingTension :=PolePar.fTension;//放卷张力
						BeltData[BeltNo.OverHang].UnreelingTension :=PolePar.fTension;//放卷张力	
						BeltData[BeltNo.OverHang].fPoleNGSizeNo:=CCD_COM.Size.fPoleNGSizeNo; 	
		                               BeltData[BeltNo.OverHang].iTabNGSizeNo:=CCD_COM.Size.iTabNGSizeNo; 	
					END_IF
					
		
						IF ABS(CCD_COM.Size.fOffsetDeg)<5 THEN
							FOR i3:=1 TO 10 BY 1 DO 
								IF i3<10 THEN 
									fOffsetDeg[11-i3]:=fOffsetDeg[10-i3];
								END_IF; 
							END_FOR; 
							fOffsetDeg[1]:=CCD_COM.Size.fOffsetDeg;		//偏移值正负要定好
						END_IF
						
						
						IF CCD_COM.Size.iFinish=1 THEN		//CCD结果OK
							BeltData[BeltNo.OverHang].iPanoramaNG:=1;
							BeltData[BeltNo.OverHang].iFinish:=CCD_COM.Size.iFinish;
							BeltData[BeltNo.OverHang].fPoleNGSizeNo:=CCD_COM.Size.fPoleNGSizeNo; 
							iAutoAuxStep3:=888;
							iNGSize:=0;
						ELSIF CCD_COM.Size.iFinish=2 THEN		//CCD结果NG
							BeltData[BeltNo.OverHang].iPanoramaNG:=2;
							BeltData[BeltNo.OverHang].iFinish:=CCD_COM.Size.iFinish;
							BeltData[BeltNo.OverHang].fPoleNGSizeNo:=CCD_COM.Size.fPoleNGSizeNo; 
							iAutoAuxStep3:=888;
							iNGSize:=iNGSize+1;	
						ELSIF CCD_COM.Size.iFinish=3 THEN		//无片
							BeltData[BeltNo.OverHang].iPanoramaNG:=3;
							BeltData[BeltNo.OverHang].iFinish:=CCD_COM.Size.iFinish;
							BeltData[BeltNo.OverHang].fPoleNGSizeNo:=CCD_COM.Size.fPoleNGSizeNo; 
							iNGSize:=iNGSize+1;	
							 
							stAlarm.arrFlowAlarm[21]:= (TRUE AND NOT ProductPar.iModeEN.bEmptyRunEN)  ;
							 
							iAutoAuxStep3:=888;
							iNGSize:=iNGSize+1;		
						END_IF	
				END_IF
			END_IF
	ELSE
		BeltData[BeltNo.OverHang].iPanoramaNG:=0;
		BeltData[BeltNo.OverHang].fPoleNGSizeNo:=CCD_COM.Size.fPoleNGSizeNo; 
		stAlarm.arrLightWarn[5]:=TRUE;//尺寸CCD检测超时，请查看！
		iAutoAuxStep3:=888;
		iNGSize:=iNGSize+1;
	END_IF
888://
;
END_CASE


///////////////////////////////////////////////////////////冲R角定位检测//////////////////////////////////////////////////////////////////
CASE iAutoAuxStep4 OF
10://
	IF arrAxisCtrl[VirAxisNo.VirMain].Status.fActPos < fRecordMouldCCDInMainPos-fRecordMouldCCDInMainPosMod+360+ProductPar.parPublic.fMainPos-10 THEN//到下个周期250度以前有效			
		IF arrAxisCtrl[VirAxisNo.VirMain].Status.fActPos>=fRecordMouldCCDInMainPos+30 THEN		
			IF CCD_COM.Chamfer.iFinish=1 THEN
				CutMark_R[0]:=FALSE;
				TabData[TabNo.MouldPhoto].fTab_OffsetM:=CCD_COM.Chamfer.fTabXOffset;
				TabData[TabNo.MouldPhoto].fTab_OffsetY:=CCD_COM.Chamfer.fTabYOffset; //20240524SJ
				iAutoAuxStep4:=888;
			ELSIF CCD_COM.Chamfer.iFinish=2 THEN
				CutMark_R[0]:=FALSE;
				TabData[TabNo.MouldPhoto].fTab_OffsetM:=CCD_COM.Chamfer.fTabXOffset;//CCD抓不到极耳时，给NG，纠偏量给1个片宽
				TabData[TabNo.MouldPhoto].fTab_OffsetY:=CCD_COM.Chamfer.fTabYOffset; //20240524SJ
				TabData[TabNo.MouldPhoto].bTabOffsetNG_M:=TRUE;
				//stAlarm.arrLightWarn[1]:=TRUE;//冲R角CCD定位检测NG，请查看！
				iAutoAuxStep4:=888;	
			ELSIF CCD_COM.Chamfer.iFinish=3 THEN
				TabData[TabNo.MouldPhoto].bTabOffsetNG_M:=TRUE;
				CutMark_R[0]:=TRUE;
				iAutoAuxStep4:=888;	
			END_IF	
		END_IF		
	ELSE			
		//TabData[TabNo.MouldPhoto].fTab_OffsetM:=PolePar.fPoleWidth;
		TabData[TabNo.MouldPhoto].fTab_OffsetM:=0;//20240524SJ
		TabData[TabNo.MouldPhoto].bTabOffsetNG_M:=TRUE;
		stAlarm.arrLightWarn[2]:=TRUE;//冲R角CCD定位检测超时，请查看！		
		iAutoAuxStep4:=889;			
	END_IF
888:
	;
END_CASE

///////////////////////////////////////////////////////////裁切定位检测////////////////////////////////////////////////////////////////////
CASE iAutoAuxStep5 OF
10://
	IF arrAxisCtrl[VirAxisNo.VirMain].Status.fActPos < fRecordCuterCCDInMainPos-fRecordCuterCCDInMainPosMod+360+ProductPar.parPublic.fMainPos-10 THEN//到下个周期250度以前有效			
		IF arrAxisCtrl[VirAxisNo.VirMain].Status.fActPos>=fRecordCuterCCDInMainPos+30 THEN		
			IF CCD_COM.Cuter.iFinish=1 THEN	
				TabData[TabNo.CuterPhoto].fTab_OffsetC:=CCD_COM.Cuter.fTabXOffset;
				InteData[InteNo.Cuter-2].fTabIntervalC:=CCD_COM.Cuter.fTabWidth;
				iAutoAuxStep5:=100;
			ELSIF CCD_COM.Cuter.iFinish=2 THEN	
				TabData[TabNo.CuterPhoto].fTab_OffsetC:=CCD_COM.Cuter.fTabXOffset;
				InteData[InteNo.Cuter-2].fTabIntervalC:=CCD_COM.Cuter.fTabWidth;//CCD抓不到极耳时，给NG，左侧相机纠偏量给1个片宽,,片宽给0
				InteData[InteNo.Cuter-2].bIntervalFail_C:=TRUE;
				TabData[TabNo.CuterPhoto].bTabOffsetNG_C:=TRUE;
				//stAlarm.arrLightWarn[3]:=TRUE;//裁切CCD定位检测NG，请查看！		
				iAutoAuxStep5:=888;
			ELSIF CCD_COM.Cuter.iFinish=3 THEN	
	                 	TabData[TabNo.CuterPhoto].fTab_OffsetC:=CCD_COM.Cuter.fTabXOffset;
				InteData[InteNo.Cuter-2].fTabIntervalC:=CCD_COM.Cuter.fTabWidth;//CCD抓不到极耳时，给NG，左侧相机纠偏量给1个片宽,,片宽给0
				InteData[InteNo.Cuter-2].bIntervalFail_C:=TRUE;
				TabData[TabNo.CuterPhoto].bTabOffsetNG_C:=TRUE;
				//stAlarm.arrLightWarn[3]:=TRUE;//裁切CCD定位检测NG，请查看！		
				iAutoAuxStep5:=888;					
			END_IF	
		END_IF		
	ELSE			
		TabData[TabNo.CuterPhoto].fTab_OffsetC:=PolePar.fPoleWidth;
		InteData[InteNo.Cuter-2].fTabIntervalC:=0;	
		InteData[InteNo.Cuter-2].bIntervalFail_C:=TRUE;
		TabData[TabNo.CuterPhoto].bTabOffsetNG_C:=TRUE;
		PolePar.AddAlarm  :=PolePar.AddAlarm +1;
		stAlarm.arrLightWarn[4]:=TRUE;//裁切CCD定位检测超时，请查看！					
		iAutoAuxStep5:=889;		
	END_IF
	
100:

	IF CCD_COM.Cuter.iFinish=1 AND ( ABS(CCD_COM.Cuter.fTabWidth-PolePar.TabWidthBace)>=0.5 ) THEN
		Production.NGFlag[15]:=TRUE;
		iTabWidth_JS:=iTabWidth_JS+1;
		iAutoAuxStep5:=200;	
	ELSE
		iTabWidth_JS:=0;
		iAutoAuxStep5:=300;	
	END_IF
200:		
	IF iTabWidth_JS >=10 AND NOT ProductPar.iModeEN.bTabWidtNGoff THEN
		stAlarm.arrFlowAlarm[41]:=TRUE;//极片来料不良，请检查
		iTabWidth_JS:=0;
	END_IF
	Production.NGFlag[15]:=FALSE;
	iAutoAuxStep5:=888;	

300:
	iTabWidth_JS:=0;
	iAutoAuxStep5:=888;	
888:
	;	
	
	
END_CASE

////////////////////////////////////////////////////////////////线扫拍照触发////////////////////////////////////////////////////////////////
ttLinePhoto(CLK:=arrAxisCtrl[VirAxisNo.VirMain].Status.fModuloSetPos>=2  
						AND arrAxisCtrl[VirAxisNo.VirMain].Status.fModuloSetPos<=6 
						AND  arrAxisCtrl[VirAxisNo.VirMain].Status.Moving 
						AND  stDriverCam.bInSync         , Q=> );
IF ttLinePhoto.Q THEN
	CCD_COM.Scan.bSendMark:=FALSE;//PLC_To_PC上位机的发送数据标志
	IF NOT ProductPar.iModeEN.bCcdTcpEN AND NOT ProductPar.iModeEN.bLineScanCCDEN  THEN//线扫OK信号
		
		CCD_COM.Scan.iResult_IO_UP:=33;//复位线扫IO结果
		CCD_COM.Scan.iResult_IO_Down:=33;
		bLineScanResult1_UP:=FALSE;
		bLineScanResult2_UP:=FALSE;
		bLineScanResult1_Down:=FALSE;
		bLineScanResult2_Down:=FALSE;
		CCD_IO.boXSPhoto:=TRUE;//自动线扫启动
		CCD_Com.iLineScanPhotoCount:=CCD_Com.iLineScanPhotoCount+1;
		IF  NOT  ProductPar.iLineScanSel THEN
	    	iAutoAuxStep11:=10;
		END_IF
		fRecordLineineScanCCDInMainPos:=arrAxisCtrl[VirAxisNo.VirMain].Status.fActPos;																								
		fRecordLineineScanCCDInMainPosMod:=arrAxisCtrl[VirAxisNo.VirMain].Status.fModuloActPos;		
	END_IF	
END_IF	

rLineScan_UPTCP(CLK:=CCD_COM.Scan.iResult_UP<>33      , Q=> );
rLineScan_DownTCP(CLK:=CCD_COM.Scan.iResult_Down<>33 , Q=> );

IF ProductPar.iLineScanSel THEN
     IF rLineScan_UPTCP.Q THEN
		 IF CCD_COM.Scan.iResult_UP<>0 THEN
		    CCD_Com.iLineScanReceiveResultCount_UP:=CCD_Com.iLineScanReceiveResultCount_UP+1;
		 END_IF
	 END_IF

     IF rLineScan_DownTCP.Q THEN
		  IF CCD_COM.Scan.iResult_Down<>0 THEN
		     CCD_Com.iLineScanReceiveResultCount_Down:=CCD_Com.iLineScanReceiveResultCount_Down+1;
		  END_IF
	 END_IF

ELSE 
			IF  rLineScanOK_UP.Q  OR rLineScanNG_UP.Q THEN
				CCD_Com.iLineScanReceiveResultCount_UP:=CCD_Com.iLineScanReceiveResultCount_UP+1;
				fDA1:=        arrAxisCtrl[VirAxisNo.VirMain].Status.fModuloActPos;
			END_IF

		    IF  rLineScanOK_Down.Q  OR rLineScanNG_Down.Q THEN
				CCD_Com.iLineScanReceiveResultCount_Down:=CCD_Com.iLineScanReceiveResultCount_Down+1;
				fDA2:=        arrAxisCtrl[VirAxisNo.VirMain].Status.fModuloActPos;
			END_IF

END_IF			
			
	IF CCD_Com.bLineScanPhotoCountClear THEN
       CCD_Com.iLineScanPhotoCount:=0;
	   CCD_Com.iLineScanReceiveResultCount_UP:=0;
	   CCD_Com.iLineScanReceiveResultCount_Down:=0;
    END_IF		
			
				
CASE iAutoAuxStep11 OF
10://
	IF arrAxisCtrl[VirAxisNo.VirMain].Status.fModuloActPos>5 AND arrAxisCtrl[VirAxisNo.VirMain].Status.fModuloActPos < ProductPar.parPublic.fMainPos-15 THEN//到下个周期判断结果前有效
			IF rLineScanOK_UP.Q THEN
				bLineScanResult1_UP:=TRUE;
			END_IF
			IF rLineScanNG_UP.Q THEN
				bLineScanResult2_UP:=TRUE;
			END_IF

			IF rLineScanOK_Down.Q THEN
				bLineScanResult1_Down:=TRUE;
			END_IF
			IF rLineScanNG_Down.Q THEN
				bLineScanResult2_Down:=TRUE;
			END_IF	
	
		IF (bLineScanResult1_UP OR bLineScanResult2_UP) AND (bLineScanResult1_Down OR bLineScanResult2_Down) THEN
			iAutoAuxStep11:=888;
		END_IF
	
	ELSIF  arrAxisCtrl[VirAxisNo.VirMain].Status.fModuloActPos > 320 THEN
		IF NOT (bLineScanResult1_UP OR bLineScanResult2_UP) AND (bLineScanResult1_Down OR bLineScanResult2_Down) THEN  //AND NOT ProductPar.iModeEN.bCcdTcpEN AND NOT ProductPar.iModeEN.bLineScanCCDEN
			stAlarm.arrFlowAlarm[25]:=TRUE;//上线扫超时报警
		END_IF
		IF (bLineScanResult1_UP OR bLineScanResult2_UP) AND NOT (bLineScanResult1_Down OR bLineScanResult2_Down) THEN//	AND NOT ProductPar.iModeEN.bCcdTcpEN AND NOT ProductPar.iModeEN.bLineScanCCDEN 
			stAlarm.arrFlowAlarm[27]:=TRUE;//下线扫超时报警
		END_IF
		iAutoAuxStep11:=886;
	END_IF
	
END_CASE

///////////////////////////////////////////////////////////CCD标定流程////////////////////////////////////////////////////////////////////
IF stSysState.iMode=3 THEN
	CASE iAutoAuxStep10 OF 
	0://
		IF 	CCD_IO.bCalibrationsDo THEN
			bChaNoPhoto:=FALSE;
			bCutNoPhoto:=FALSE;			
			iAutoAuxStep10:=10;
		ELSIF NOT CCD_IO.bCalibrationsDo AND CCD_IO.bCalibrationsDo_Cha AND NOT CCD_IO.bCalibrationsDo_Cut THEN
			bChaNoPhoto:=FALSE;
			bCutNoPhoto:=TRUE;
			iAutoAuxStep10:=10;
		ELSIF NOT CCD_IO.bCalibrationsDo AND NOT CCD_IO.bCalibrationsDo_Cha AND CCD_IO.bCalibrationsDo_Cut THEN
			bChaNoPhoto:=TRUE;
			bCutNoPhoto:=FALSE;			
			iAutoAuxStep10:=10;
		END_IF
	10://
		CCD_IO.bDemRuning:=TRUE;
		CCD_COM.iDemCount:=1;//是否需要延时
		iAutoAuxStep10:=20;
	20://
		IF NOT bChaNoPhoto THEN
			CCD_COM.iDemResult_Cha:=0;
			CCD_IO.hmiChamferPhoto:=TRUE;
		END_IF
		IF NOT bCutNoPhoto THEN
			CCD_COM.iDemResult_Cut:=0;
			CCD_IO.hmiCuterPhoto:=TRUE;
		END_IF	
		iAutoAuxStep10:=30;
	30://
		IF tonAuto[17].Q THEN
			CCD_IO.hmiChamferPhoto:=FALSE;
			CCD_IO.hmiCuterPhoto:=FALSE;
			tonAuto[18].IN:=FALSE;
			iAutoAuxStep10:=40;
		END_IF
	40://
		IF (bChaNoPhoto  OR CCD_COM.iDemResult_Cha=1) AND (bCutNoPhoto OR CCD_COM.iDemResult_Cut=1) THEN
			tonAuto[18].IN:=FALSE;
			iAutoAuxStep10:=50;
		ELSIF (NOT bChaNoPhoto  AND CCD_COM.iDemResult_Cha=2) OR (NOT bCutNoPhoto AND CCD_COM.iDemResult_Cut=2) THEN
			tonAuto[18].IN:=FALSE;
			iAutoAuxStep10:=999;
		ELSE
			IF NOT tonAuto[18].Q THEN
				tonAuto[18].IN:=TRUE;
			ELSE
				tonAuto[18].IN:=FALSE;
				iAutoAuxStep10:=999;
			END_IF
		END_IF
	50://
		arrAxisCtrl[AxisNo.DriverDDR].Cmd.fPositon_of_Abs:=arrAxisCtrl[AxisNo.DriverDDR].Status.fActPos+FC_LengthToAngle(CCD_COM.fDemLength,PolePar.Machine.fMQDriverDiameter);
		arrAxisPar[AxisNo.DriverDDR].fVelocity_of_Abs:=5;
		arrAxisCtrl[AxisNo.DriverDDR].Cmd.bMoveAbs:=TRUE;
		iAutoAuxStep10:=60;
	60://
		IF arrAxisCtrl[AxisNo.DriverDDR].Status.Moving THEN
			CCD_COM.iDemCount:=2;
			iAutoAuxStep10:=70;
		END_IF
	70://
		IF NOT arrAxisCtrl[AxisNo.DriverDDR].Cmd.bMoveAbs AND arrAxisCtrl[AxisNo.DriverDDR].Status.NoMoving THEN
			iAutoAuxStep10:=80;
		END_IF
	80://
		IF NOT bChaNoPhoto THEN
			CCD_COM.iDemResult_Cha:=0;
			CCD_IO.hmiChamferPhoto:=TRUE;
		END_IF
		IF NOT bCutNoPhoto THEN
			CCD_COM.iDemResult_Cut:=0;
			CCD_IO.hmiCuterPhoto:=TRUE;
		END_IF	
		iAutoAuxStep10:=90;		
	90://
		IF tonAuto[17].Q THEN
			CCD_IO.hmiChamferPhoto:=FALSE;
			CCD_IO.hmiCuterPhoto:=FALSE;
			tonAuto[18].IN:=FALSE;
			iAutoAuxStep10:=100;
			arrAxisCtrl[AxisNo.DriverDDR].Cmd.fPositon_of_Abs:=arrAxisCtrl[AxisNo.DriverDDR].Status.fActPos-FC_LengthToAngle(CCD_COM.fDemLength,PolePar.Machine.fMQDriverDiameter);
			arrAxisPar[AxisNo.DriverDDR].fVelocity_of_Abs:=20;
			arrAxisCtrl[AxisNo.DriverDDR].Cmd.bMoveAbs:=TRUE;			
		END_IF	
	100://
		IF (bChaNoPhoto  OR CCD_COM.iDemResult_Cha=1) AND (bCutNoPhoto OR CCD_COM.iDemResult_Cut=1) THEN
			tonAuto[18].IN:=FALSE;
			iAutoAuxStep10:=666;
		ELSIF (NOT bChaNoPhoto  AND CCD_COM.iDemResult_Cha=2) OR (NOT bCutNoPhoto AND CCD_COM.iDemResult_Cut=2) THEN
			tonAuto[18].IN:=FALSE;
			iAutoAuxStep10:=999;
		ELSE
			IF NOT tonAuto[18].Q THEN
				tonAuto[18].IN:=TRUE;
			ELSE
				tonAuto[18].IN:=FALSE;
				iAutoAuxStep10:=999;
			END_IF
		END_IF	
	666://
		CCD_COM.iDemCount:=999;
		IF NOT bChaNoPhoto THEN
			CCD_IO.bCalibrationsDone_Cha:=TRUE;
		END_IF
		IF NOT bCutNoPhoto THEN
			CCD_IO.bCalibrationsDone_Cut:=TRUE;
		END_IF
		CCD_IO.bDemRuning:=FALSE;
		IF NOT arrAxisCtrl[AxisNo.DriverDDR].Cmd.bMoveAbs AND arrAxisCtrl[AxisNo.DriverDDR].Status.NoMoving THEN	
			iAutoAuxStep10:=0;
		END_IF
	999://
		CCD_COM.iDemCount:=999;
		IF NOT bChaNoPhoto THEN
			CCD_IO.bCalibrationsFals_Cha:=TRUE;
		END_IF
		IF NOT bCutNoPhoto THEN
			CCD_IO.bCalibrationsFals_Cut:=TRUE;
		END_IF
		CCD_IO.bDemRuning:=FALSE;	
		IF NOT arrAxisCtrl[AxisNo.DriverDDR].Cmd.bMoveAbs AND arrAxisCtrl[AxisNo.DriverDDR].Status.NoMoving THEN	
			iAutoAuxStep10:=0;
		END_IF
	END_CASE
ELSE
	CCD_COM.iDemCount:=999;
	CCD_IO.bDemRuning:=FALSE;
	iAutoAuxStep10:=0;		
END_IF


	(*
////////////////////////////////////////////////////////////////线扫拍照触发////////////////////////////////////////////////////////////////
ttLinePhoto(CLK:=arrAxisCtrl[VirAxisNo.VirMain].Status.fModuloSetPos>=2  
						AND arrAxisCtrl[VirAxisNo.VirMain].Status.fModuloSetPos<=6 
						AND  arrAxisCtrl[VirAxisNo.VirMain].Status.Moving 
						AND  stDriverCam.bInSync         , Q=> );
IF ttLinePhoto.Q THEN
	IF NOT ProductPar.iModeEN.bCcdTcpEN   THEN//线扫OK信号  //AND NOT ProductPar.iModeEN.bLineScanCCDEN
			IF BeltData[BeltNo.LineScanUp].iJumpCutNG=1 AND BeltData[BeltNo.LineScanUp+1].iJumpCutNG=1 AND BeltData[BeltNo.LineScanUp].fPoleNGSizeNo=30 THEN
				CCD_IO.hmiXSPhotoUp:=TRUE;//自动线扫启动
				CCD_COM.Scan.stPoleNoUp:=BeltData[BeltNo.LineScanUp].stPoleNo;			
			END_IF
			IF BeltData[BeltNo.LineScanDown].iJumpCutNG=1 AND BeltData[BeltNo.LineScanDown+1].iJumpCutNG=1 AND BeltData[BeltNo.LineScanDown].fPoleNGSizeNo=30 THEN
				CCD_IO.hmiXSPhotoDown:=TRUE;//自动线扫启动
				CCD_COM.Scan.stPoleNoDown:=BeltData[BeltNo.LineScanDown].stPoleNo;		
			END_IF		
			fRecordLineineScanCCDInMainPos:=arrAxisCtrl[VirAxisNo.VirMain].Status.fActPos;																								
			fRecordLineineScanCCDInMainPosMod:=arrAxisCtrl[VirAxisNo.VirMain].Status.fModuloActPos;	
	END_IF	
END_IF	
	*)


	
	
	
	
	(*


CASE iAutoAuxStep2 OF
100://
	IF NOT ProductPar.iModeEN.bEmptyRunEN THEN
		bMethodTenBufferEnable:=TRUE;
		iAutoAuxStep2:=200;
	ELSE
		bMethodTenBufferDisEnable:=TRUE;
		iAutoAuxStep2:=300;
	END_IF	
200://
	IF NOT bMethodTenBufferEnable THEN
		iAutoAuxStep2:=666;
	END_IF
300://
	IF NOT bMethodTenBufferDisEnable THEN
		iAutoAuxStep2:=350;
	END_IF
350://	
	arrCyCtrl[CYNo.DriverPressDDR].Cmd.bOFF:=TRUE;
	IF arrCyCtrl[CYNo.DriverPressDDR].Status.OFFState THEN
		iAutoAuxStep2:=666;
	END_IF
END_CASE
	
	*)
END_ACTION

ACTION F0512CarryAuto:
////////////////////////////////////////////////////////////////送片模式选择////////////////////////////////////////////////////////////////
IF ProductPar.iModeEN.bP2PartEN THEN
	iPoleCarryEver:=3;
ELSE
	iPoleCarryEver:=ProductPar.iModeEN.iCarryPoleMode;
END_IF
////////////////////////////////////////////////////////////////料况转化////////////////////////////////////////////////////////////////
bBelt_1[1]:=BeltData[BeltNo.SubBelt1].bHavePole;
bBelt_2[1]:=BeltData[BeltNo.SubBelt1-1].bHavePole;
bBelt_1[2]:=BeltData[BeltNo.SubBelt2].bHavePole;
bBelt_2[2]:=BeltData[BeltNo.SubBelt2-1].bHavePole;
bBelt_1[3]:=BeltData[BeltNo.SubBelt3].bHavePole;
bBelt_2[3]:=BeltData[BeltNo.SubBelt3-1].bHavePole;
////////////////////////////////////////////////////////////////送片皮带要料逻辑(皮带耦合,无料统计)    纯靠料况////////////////////////////////////////////////////////////////

bBelt_NO1:=bBelt_2[1] AND NOT bBelt_1[1] AND (   (bBelt_1[2] AND bBelt_1[3])  ) ;
bBelt_NO2:=bBelt_2[2] AND NOT bBelt_1[2] AND (  (bBelt_1[1] AND  bBelt_1[3])   ) ; 
bBelt_NO3:= ( bBelt_2[3] AND NOT bBelt_1[3] AND (   (bBelt_1[1] AND bBelt_1[2])  )  ) OR
			( bBelt_2[3] AND bBelt_1[3] AND (BeltData[BeltNo.SubBelt3].stPoleNo=''AND NOT ProductPar.iModeEN.bCcdTcpEN AND NOT ProductPar.iModeEN.bSizeCCDEN)
			AND (   (bBelt_1[1] AND bBelt_1[2]) ) ) ;


IF iPoleCarryEver=3 THEN
	bBelt3Need:=NOT BeltData[BeltNo.SubBelt3].bHavePole OR (BeltData[BeltNo.SubBelt3].bHavePole AND (BeltData[BeltNo.SubBelt3].stPoleNo=''AND NOT ProductPar.iModeEN.bCcdTcpEN AND NOT ProductPar.iModeEN.bSizeCCDEN) ) OR ProductPar.iModeEN.bP2PartEN;					
	bBelt2Need:=NOT BeltData[BeltNo.SubBelt2].bHavePole OR	 bBelt3Need;	
	
	IF bBelt_1[1] AND bBelt_1[2] AND (bBelt_1[3] AND (BeltData[BeltNo.SubBelt3].stPoleNo<>'' OR ProductPar.iModeEN.bCcdTcpEN OR ProductPar.iModeEN.bSizeCCDEN)) AND NOT ProductPar.iModeEN.bP2PartEN THEN
		iPoleNoHaveA:=0;
	ELSIF (bBelt_NO1 OR bBelt_NO2  OR bBelt_NO3 ) AND NOT ProductPar.iModeEN.bP2PartEN THEN
		iPoleNoHaveA:=1;
	ELSE
		iPoleNoHaveA:=2;	
	END_IF
ELSIF iPoleCarryEver=2 THEN
	bBelt3Need:=FALSE;
	bBelt2Need:=NOT BeltData[BeltNo.SubBelt2].bHavePole OR	 bBelt3Need;
	
	IF bBelt_1[1] AND bBelt_1[2]  AND NOT ProductPar.iModeEN.bP2PartEN   THEN
		iPoleNoHaveA:=0;
	ELSIF(
             (  bBelt_2[1] AND NOT bBelt_1[1] AND (  bBelt_1[2]  )   ) OR
			 (  bBelt_2[2] AND NOT bBelt_1[2] AND (  bBelt_1[1]  )   )
            )  AND NOT ProductPar.iModeEN.bP2PartEN  THEN
		iPoleNoHaveA:=1;
	ELSE
		iPoleNoHaveA:=2;	
	END_IF	
ELSE
	bBelt3Need:=FALSE;
	bBelt2Need:=FALSE OR	bBelt3Need;
	IF bBelt_1[1]  AND NOT ProductPar.iModeEN.bP2PartEN   THEN
		iPoleNoHaveA:=0;
	ELSIF ( bBelt_2[1] AND NOT bBelt_1[1] )  AND NOT ProductPar.iModeEN.bP2PartEN       THEN
		iPoleNoHaveA:=1;
	ELSE
		iPoleNoHaveA:=2;	
	END_IF							
END_IF

//取料位置有无片信号清理
IF rMQUse[11].Q THEN//叠台1
	BeltData[BeltNo.SubBelt1].bHavePole:=FALSE ;	
END_IF
IF rMQUse[12].Q THEN//叠台2
	BeltData[BeltNo.SubBelt2].bHavePole:=FALSE ;	
END_IF
IF rMQUse[13].Q THEN//叠台3
	BeltData[BeltNo.SubBelt3].bHavePole:=FALSE ;	
END_IF

(*****************减少取片等待时间*****************)
CASE iAutoAuxStep9 OF	
	100:
		tMQUse[1](IN:=FALSE , PT:=T#5S , Q=> , ET=> );
		IF iPartSelect=2 THEN
			iAutoAuxStep9:=200;//负极
		ELSE
			iAutoAuxStep9:=200;//300;//正极 20240509 CF
		END_IF
	200://负极不判断叠片主轴位置
		tMQUse[1](IN:=TRUE , PT:=T#5S , Q=> , ET=> );
		IF (InterPart.M1LockReady OR InterPart.M1JumpReady) AND (InterPart.M2LockReady OR InterPart.M2JumpReady) AND
			(InterPart.M3LockReady OR InterPart.M3JumpReady) THEN//OR tMQUse[1].Q 
			iAutoAuxStep9:=400;
		END_IF
	300://正极判断叠片主轴位置
		tMQUse[1](IN:=TRUE , PT:=T#5S , Q=> , ET=> );
		IF InterPart.M1LockReady AND InterPart.M2LockReady AND InterPart.M3LockReady THEN
			IF ABS(D_Sys.fM1MainSetPos-D_Sys.fM2MainSetPos)<1 AND ABS(D_Sys.fM1MainSetPos-D_Sys.fM3MainSetPos)<1
				AND ABS(D_Sys.fM2MainSetPos-D_Sys.fM3MainSetPos)<1 THEN
				iAutoAuxStep9:=400;//三个叠台同步
			END_IF
		ELSIF InterPart.M1LockReady AND InterPart.M2LockReady AND InterPart.M3JumpReady THEN
			IF ABS(D_Sys.fM1MainSetPos-D_Sys.fM2MainSetPos)<1 THEN
				iAutoAuxStep9:=400;// 1、2叠台同步
			END_IF
		ELSIF InterPart.M1LockReady AND InterPart.M2JumpReady AND InterPart.M3LockReady THEN
			IF ABS(D_Sys.fM1MainSetPos-D_Sys.fM3MainSetPos)<1 THEN
				iAutoAuxStep9:=400;//1、3叠台同步
			END_IF
		ELSIF InterPart.M1JumpReady AND InterPart.M2LockReady AND InterPart.M3LockReady THEN
			IF ABS(D_Sys.fM2MainSetPos-D_Sys.fM3MainSetPos)<1 THEN
				iAutoAuxStep9:=400;//2、3叠台同步
			END_IF
		ELSIF (InterPart.M1LockReady AND InterPart.M2JumpReady AND InterPart.M3JumpReady) 
				OR (InterPart.M1JumpReady AND InterPart.M2LockReady AND InterPart.M3JumpReady)
				OR (InterPart.M1JumpReady AND InterPart.M2JumpReady AND InterPart.M3LockReady) OR tMQUse[1].Q THEN
				iAutoAuxStep9:=400;//单个叠台
		END_IF
	400://允许取片信号   
		arrModPos[K10]:='';
		IF 	InterPart.M1LockReady AND (BeltData[BeltNo.SubBelt1].stPoleNo<>'' OR ProductPar.iModeEN.bCcdTcpEN OR ProductPar.iModeEN.bSizeCCDEN)  AND NOT bBelt1Taking THEN
			arrModPos[K10]:= CONCAT( arrModPos[K10], CONCAT( '     1#: ',REAL_TO_STRING(D_Sys.fM1MainSetPos)));	
			bMA10:=TRUE;
			iAutoAuxStep6:=10;
		END_IF
		IF 	InterPart.M2LockReady AND (BeltData[BeltNo.SubBelt2].stPoleNo<>''OR ProductPar.iModeEN.bCcdTcpEN OR ProductPar.iModeEN.bSizeCCDEN) AND NOT bBelt2Taking THEN
			arrModPos[K10]:= CONCAT( arrModPos[K10], CONCAT( '     2#: ',REAL_TO_STRING(D_Sys.fM2MainSetPos)));	
			bMA10:=TRUE;
			iAutoAuxStep7:=10;
		END_IF	
		IF 	InterPart.M3LockReady AND (BeltData[BeltNo.SubBelt3].stPoleNo<>''OR ProductPar.iModeEN.bCcdTcpEN OR ProductPar.iModeEN.bSizeCCDEN) AND NOT bBelt3Taking THEN
			arrModPos[K10]:= CONCAT( arrModPos[K10], CONCAT( '     3#: ',REAL_TO_STRING(D_Sys.fM3MainSetPos)));	
			bMA10:=TRUE;
			iAutoAuxStep8:=10;
		END_IF
		
		IF bMA10 THEN
			K10:=K10+1;
			IF K10>500 THEN
				K10:=1;
				MEMSET(ADR(arrModPos),0,SIZEOF(arrModPos));			
			END_IF
		   bMA10:=FALSE;
		END_IF
		
		iAutoAuxStep9:=666;	
END_CASE


///////////////////////////////////////////////////////////允许1叠台取料信号复位///////////////////////////////////////////////////////////////////20221101BYSJ
rtBelt1TakingReset1(CLK:=arrAxisCtrl[VirAxisNo.VirMain].Status.fModuloActPos>=10  AND   arrAxisCtrl[VirAxisNo.VirMain].Status.fModuloActPos<=20  AND 
                                      arrAxisCtrl[VirAxisNo.VirMain].Status.fSetVelo>=0.5          AND    bSubBelt1fratio      , Q=> );
rtBelt1TakingReset2(CLK:=arrAxisCtrl[VirAxisNo.VirMain].Status.fModuloActPos>=10  AND   arrAxisCtrl[VirAxisNo.VirMain].Status.fModuloActPos<=20  AND 
                                      arrAxisCtrl[VirAxisNo.VirMain].Status.fSetVelo>=0.5          AND    bSubBelt2fratio      , Q=> );									  
rtBelt1TakingReset3(CLK:=arrAxisCtrl[VirAxisNo.VirMain].Status.fModuloActPos>=10  AND   arrAxisCtrl[VirAxisNo.VirMain].Status.fModuloActPos<=20  AND 
                                      arrAxisCtrl[VirAxisNo.VirMain].Status.fSetVelo>=0.5          AND    bSubBelt3fratio      , Q=> );								  									  
IF  rtBelt1TakingReset1.Q THEN
	  InterPart.M1Allow:=FALSE;
      iAutoAuxStep6:=886;
END_IF	  
IF  rtBelt1TakingReset2.Q THEN
	  InterPart.M2Allow:=FALSE;
      iAutoAuxStep7:=886;
END_IF	  	  
IF  rtBelt1TakingReset3.Q THEN
	  InterPart.M3Allow:=FALSE;
      iAutoAuxStep8:=886;
END_IF	  



